# B&R Automation Studio project HealthCareDemo (part 4)

#### Types.typ
```iecst
TYPE
	Vis6D_typ : 	STRUCT
		Cmd : Vis6DCmd_typ;
		Par : Pars6D_typ;
		Status : Vis6DStatus_typ;
		TableData : VisTableData_typ;
		Limits : Vis6DLimits_typ;
	END_STRUCT;
	Vis6DCmd_typ : 	STRUCT
		ErrorReset : BOOL;
		Power : BOOL;
		AsmStop : BOOL;
		ShStop : BOOL;
		AsmHalt : BOOL;
		ShHalt : BOOL;
		AsmResume : BOOL;
		ShResume : BOOL;
		ShuttleID : UINT;
		RecoverShuttle : BOOL;
		MoveLinear : BOOL;
		MoveArc : BOOL;
		MoveShort : BOOL;
		MoveAsync : BOOL;
		Move6DOF : BOOL;
		AsmLevitation : BOOL;
		ShLevitation : BOOL;
		AsmBuffer : BOOL;
		ShBuffer : BOOL;
		Reboot : BOOL;
		ShRecover : BOOL;
	END_STRUCT;
	Vis6DStatus_typ : 	STRUCT
		AsmStatus : AsmStatus_typ;
		AllShuttlesFound : BOOL;
		StatusMessage : STRING[80];
		CurrentState : STRING[80];
		ErrorID : DINT;
		SelectedShuttleIDString : STRING[80];
		MovementActive : BOOL;
		ShuttleBuffer : VisShuttleBufferStatus_typ;
		ErrorText : STRING[80];
	END_STRUCT;
	VisShuttleBufferStatus_typ : 	STRUCT
		ShuttleID : UINT;
		State : STRING[80];
		NumberOfCommands : UINT;
	END_STRUCT;
	VisTableData_typ : 	STRUCT
		Async : VisAsyncTable_typ;
		ShuttleStatus : VisShuttleStatusTable_typ;
	END_STRUCT;
	VisAsyncTable_typ : 	STRUCT
		TargetXArray : ARRAY[0..rdiMAX_ASYNC_SHUTTLES_M1]OF REAL;
		TargetYArray : ARRAY[0..rdiMAX_ASYNC_SHUTTLES_M1]OF REAL;
		ShuttleIDArray : ARRAY[0..rdiMAX_ASYNC_SHUTTLES_M1]OF UINT;
	END_STRUCT;
	VisShuttleStatusTable_typ : 	STRUCT
		ShuttleID : ARRAY[0..MAX_NUM_SHUTTLES_M1]OF UINT;
		ShuttleIDString : ARRAY[0..MAX_NUM_SHUTTLES_M1]OF STRING[80];
		ShuttleStateText : ARRAY[0..MAX_NUM_SHUTTLES_M1]OF STRING[80];
		X : ARRAY[0..MAX_NUM_SHUTTLES_M1]OF REAL;
		Y : ARRAY[0..MAX_NUM_SHUTTLES_M1]OF REAL;
		Z : ARRAY[0..MAX_NUM_SHUTTLES_M1]OF REAL;
		Rx : ARRAY[0..MAX_NUM_SHUTTLES_M1]OF REAL;
		Ry : ARRAY[0..MAX_NUM_SHUTTLES_M1]OF REAL;
		Rz : ARRAY[0..MAX_NUM_SHUTTLES_M1]OF REAL;
	END_STRUCT;
END_TYPE

(*Insert your comment here.*)

TYPE
	Vis6DRealMinMax_typ : 	STRUCT
		Min : REAL;
		Max : REAL;
	END_STRUCT;
	Vis6DLimits_typ : 	STRUCT
		Linear : Vis6DLimitsLinear_typ;
		Arc : Vis6DLimitsArc_typ;
		Short : Vis6DLimitsShort_typ;
		SixDOF : Vis6DLimits6DOF_typ;
		Async : Vis6DLimitsAsync_typ;
	END_STRUCT;
	Vis6DLimitsLinear_typ : 	STRUCT
		X : Vis6DRealMinMax_typ;
		Y : Vis6DRealMinMax_typ;
		Velocity : Vis6DRealMinMax_typ;
		EndVelocity : Vis6DRealMinMax_typ;
		Acceleration : Vis6DRealMinMax_typ;
	END_STRUCT;
	Vis6DLimitsArc_typ : 	STRUCT
		AngleX : Vis6DRealMinMax_typ;
		AngleY : Vis6DRealMinMax_typ;
		Angle : Vis6DRealMinMax_typ;
		RadiusX : Vis6DRealMinMax_typ;
		RadiusY : Vis6DRealMinMax_typ;
		Radius : Vis6DRealMinMax_typ;
		Velocity : Vis6DRealMinMax_typ;
		EndVelocity : Vis6DRealMinMax_typ;
		Acceleration : Vis6DRealMinMax_typ;
	END_STRUCT;
	Vis6DLimitsShort_typ : 	STRUCT
		CenterX : Vis6DRealMinMax_typ;
		CenterY : Vis6DRealMinMax_typ;
		Z : Vis6DRealMinMax_typ;
		Rx : Vis6DRealMinMax_typ;
		Ry : Vis6DRealMinMax_typ;
		Rz : Vis6DRealMinMax_typ;
		VelZ : Vis6DRealMinMax_typ;
		VelRx : Vis6DRealMinMax_typ;
		VelRy : Vis6DRealMinMax_typ;
		VelRz : Vis6DRealMinMax_typ;
	END_STRUCT;
	Vis6DLimits6DOF_typ : 	STRUCT
		X : Vis6DRealMinMax_typ;
		Y : Vis6DRealMinMax_typ;
		Velocity : Vis6DRealMinMax_typ;
		Acceleration : Vis6DRealMinMax_typ;
		Z : Vis6DRealMinMax_typ;
		Rx : Vis6DRealMinMax_typ;
		Ry : Vis6DRealMinMax_typ;
		Rz : Vis6DRealMinMax_typ;
		VelZ : Vis6DRealMinMax_typ;
		VelRx : Vis6DRealMinMax_typ;
		VelRy : Vis6DRealMinMax_typ;
		VelRz : Vis6DRealMinMax_typ;
	END_STRUCT;
	Vis6DLimitsAsync_typ : 	STRUCT
		Velocity : Vis6DRealMinMax_typ;
		Acceleration : Vis6DRealMinMax_typ;
		X : Vis6DRealMinMax_typ;
		Y : Vis6DRealMinMax_typ;
	END_STRUCT;
END_TYPE
```

#### Variables.var
```iecst
VAR
	i : UINT;
	Core : rdi6DCore;
	Pars : Pars6D_typ;
	Vis : Vis6D_typ := (Limits:=(Linear:=(X:=(Min:=0.0,Max:=0.42),Y:=(Min:=0.0,Max:=0.18),Velocity:=(Min:=0.0,Max:=1.0),EndVelocity:=(Min:=0.0,Max:=1.0),Acceleration:=(Min:=0.0,Max:=10.0)),Arc:=(AngleX:=(Min:=0.0,Max:=0.42),AngleY:=(Min:=0.0,Max:=0.18),Angle:=(Min:=0.0,Max:=6.28319),RadiusX:=(Min:=0.0,Max:=0.42),RadiusY:=(Min:=0.0,Max:=0.18),Radius:=(Min:=0.0,Max:=0.1),Velocity:=(Min:=0.0,Max:=1.0),EndVelocity:=(Min:=0.0,Max:=1.0),Acceleration:=(Min:=0.0,Max:=10.0)),Short:=(CenterX:=(Min:=0.0,Max:=0.42),CenterY:=(Min:=0.0,Max:=0.18),Z:=(Min:=0.0,Max:=0.003),Rx:=(Min:=0.0,Max:=0.0872665),Ry:=(Min:=0.0,Max:=0.0872665),Rz:=(Min:=0.0,Max:=0.226893),VelZ:=(Min:=0.0,Max:=0.15),VelRx:=(Min:=0.0,Max:=0.1),VelRy:=(Min:=0.0,Max:=0.1),VelRz:=(Min:=0.0,Max:=0.3)),SixDOF:=(X:=(Min:=0.0,Max:=0.42),Y:=(Min:=0.0,Max:=0.18),Velocity:=(Min:=0.0,Max:=1.0),Acceleration:=(Min:=0.0,Max:=10.0),Z:=(Min:=0.0,Max:=0.003),Rx:=(Min:=0.0,Max:=0.0872665),Ry:=(Min:=0.0,Max:=0.0872665),Rz:=(Min:=0.0,Max:=0.226893),VelZ:=(Min:=0.0,Max:=0.15),VelRx:=(Min:=0.0,Max:=0.1),VelRy:=(Min:=0.0,Max:=0.1),VelRz:=(Min:=0.0,Max:=0.3)),Async:=(Velocity:=(Min:=0.0,Max:=1.0),Acceleration:=(Min:=0.0,Max:=10.0),X:=(Min:=0.0,Max:=0.42),Y:=(Min:=0.0,Max:=0.18))));
	TestStart : BOOL;
	ShState : McAcp6DShStateEnum;
	ShStatusTexts : ARRAY[0..15] OF STRING[80] := ['UNDETECTED','DISCOVERING','LANDED','IDLING','DISABLED','MOTION','WAIT','STOPPING','OBSTACLE','HOLD','STOPPED',3(''),'ERROR','RESERVED'];
	ShBufferStateTexts : ARRAY[0..1] OF STRING[80] := ['OPEN','BLOCKED'];
	StringPlacehold : STRING[80];
END_VAR
```

#### Main.st
```iecst
PROGRAM _INIT
	Core.Parameters := ADR(Pars);
	Core.AsmRef := ADR(g6dAssembly);
	Core.Enable := TRUE;
	ShState;
	TestStart := TRUE;

	Vis.Cmd.ShuttleID := 1;
	//

	Vis.Par.Linear.Position.X := 0.12;		// m
	Vis.Par.Linear.Position.Y := 0.12;		// m
	Vis.Par.Linear.Velocity := 1.0;			// m/s
	Vis.Par.Linear.EndVelocity := 0.0;		// m/s
	Vis.Par.Linear.Acceleration := 10.0;	// m/s^2

	Vis.Par.Arc.Radius.Position.X := 0.12;	// m
	Vis.Par.Arc.Radius.Position.Y := 0.12; // m
	Vis.Par.Arc.Radius.Radius := 0.0;		// m
	Vis.Par.Arc.Angular.Center.X := 0.12;	// m
	Vis.Par.Arc.Angular.Center.Y := 0.12;	// m
	Vis.Par.Arc.Angular.Angle := 0.0;		// rad
	Vis.Par.Arc.Velocity := 1.0;			// m/s
	Vis.Par.Arc.EndVelocity := 0.0;			// m/s
	Vis.Par.Arc.Acceleration := 10.0;		// m/s^2

	Vis.Par.ShortAxis.Rotation.Center.X := 0.18;	// m
	Vis.Par.ShortAxis.Rotation.Center.Y := 0.18;	// m
	Vis.Par.ShortAxis.Position.Z := 0.001;			// m
	Vis.Par.ShortAxis.Velocity.Z := 0.002;			// m/s
	Vis.Par.ShortAxis.Velocity.Rx := 0.0873;		// rad/s
	Vis.Par.ShortAxis.Velocity.Ry := 0.0873;		// rad/s
	Vis.Par.ShortAxis.Velocity.Rz := 0.0873;		// rad/s

	Vis.Par.SixDOF.InPlane.Position.X := 0.12;		// m
	Vis.Par.SixDOF.InPlane.Position.Y := 0.12;		// m
	Vis.Par.SixDOF.ShortAxis.Position.Z := 0.001;	// m
	Vis.Par.SixDOF.InPlane.Velocity := 1.0;			// m/s
	Vis.Par.SixDOF.InPlane.Acceleration := 10.0;	// m/s^2
	Vis.Par.SixDOF.ShortAxis.Velocity.Z := 0.002;	// m/s
	Vis.Par.SixDOF.ShortAxis.Velocity.Rx := 0.0873;	// rad/s
	Vis.Par.SixDOF.ShortAxis.Velocity.Ry := 0.0873;	// rad/s
	Vis.Par.SixDOF.ShortAxis.Velocity.Rz := 0.0873;	// rad/s

	Vis.Par.Async.Velocity := 0.5;		// m/s
	Vis.Par.Async.Acceleration := 5.0;	// m/s^2

END_PROGRAM

PROGRAM _CYCLIC
	(* Insert code here *)
	gFB;

	IF TestStart THEN
		Vis.Cmd.ShuttleID := STRING_TO_UINT(Vis.Status.SelectedShuttleIDString);

		Core.Power := Vis.Cmd.Power;
		Core.ShuttleID := Vis.Cmd.ShuttleID;
		Core.ErrorReset := Vis.Cmd.ErrorReset;

		Core.MoveLinear := Vis.Cmd.MoveLinear;
		Core.MoveArc := Vis.Cmd.MoveArc;
		Core.MoveShort := Vis.Cmd.MoveShort;
		Core.Move6DOF := Vis.Cmd.Move6DOF;
		Core.MoveAsync := Vis.Cmd.MoveAsync;

		Core.AsmStop := Vis.Cmd.AsmStop;
		Core.AsmHalt := Vis.Cmd.AsmHalt;
		Core.AsmResume := Vis.Cmd.AsmResume;

		Core.ShStop := Vis.Cmd.ShStop;
		Core.ShHalt := Vis.Cmd.ShHalt;
		Core.ShResume := Vis.Cmd.ShResume;

		Core.AsmLevitation := Vis.Cmd.AsmLevitation;
		Core.ShLevitation := Vis.Cmd.ShLevitation;
		Core.AsmBuffer := Vis.Cmd.AsmBuffer;
		Core.ShBuffer := Vis.Cmd.ShBuffer;

		Core.Reboot := Vis.Cmd.Reboot;
		Core.ShRecover := Vis.Cmd.ShRecover;

		FOR i := 0 TO rdiMAX_ASYNC_SHUTTLES_M1 DO
			Vis.Par.Async.ShuttleTable[i].ShuttleID := Vis.TableData.Async.ShuttleIDArray[i];
			Vis.Par.Async.ShuttleTable[i].X := Vis.TableData.Async.TargetXArray[i];
			Vis.Par.Async.ShuttleTable[i].Y := Vis.TableData.Async.TargetYArray[i];
		END_FOR

		FOR i := 0 TO MAX_NUM_SHUTTLES_M1 DO
			Vis.TableData.ShuttleStatus.ShuttleID[i] := Core.ShuttleArray[i].ShuttleID;

			Vis.TableData.ShuttleStatus.ShuttleIDString[i] := '{"value":"';
			StringPlacehold := UINT_TO_STRING(Core.ShuttleArray[i].ShuttleID);
			Vis.TableData.ShuttleStatus.ShuttleIDString[i] := CONCAT(Vis.TableData.ShuttleStatus.ShuttleIDString[i], StringPlacehold);
			Vis.TableData.ShuttleStatus.ShuttleIDString[i] := CONCAT(Vis.TableData.ShuttleStatus.ShuttleIDString[i], '","text":"');
			StringPlacehold := UINT_TO_STRING(Core.ShuttleArray[i].ShuttleID);
			Vis.TableData.ShuttleStatus.ShuttleIDString[i] := CONCAT(Vis.TableData.ShuttleStatus.ShuttleIDString[i], StringPlacehold);
			Vis.TableData.ShuttleStatus.ShuttleIDString[i] := CONCAT(Vis.TableData.ShuttleStatus.ShuttleIDString[i], '"}');

			Vis.TableData.ShuttleStatus.ShuttleStateText[i] := ShStatusTexts[Core.ShuttleArray[i].State];

			Vis.TableData.ShuttleStatus.X[i] := Core.ShuttleArray[i].Position.X;
			Vis.TableData.ShuttleStatus.Y[i] := Core.ShuttleArray[i].Position.Y;
			Vis.TableData.ShuttleStatus.Z[i] := Core.ShuttleArray[i].Position.Z;
			Vis.TableData.ShuttleStatus.Rx[i] := Core.ShuttleArray[i].Position.Rx;
			Vis.TableData.ShuttleStatus.Ry[i] := Core.ShuttleArray[i].Position.Ry;
			Vis.TableData.ShuttleStatus.Rz[i] := Core.ShuttleArray[i].Position.Rz;

		END_FOR

		brsmemcpy(ADR(Pars), ADR(Vis.Par), SIZEOF(Pars6D_typ));

		(* Copy Statuses *)
		brsmemcpy(ADR(Vis.Status.AsmStatus), ADR(Core.AsmStatus), SIZEOF(AsmStatus_typ));
		brsmemcpy(ADR(Vis.Status.StatusMessage), ADR(Core.StatusMessage), SIZEOF(Vis.Status.StatusMessage));
		brsmemcpy(ADR(Vis.Status.CurrentState), ADR(Core.CurrentState), SIZEOF(Vis.Status.CurrentState));

		Vis.Status.AllShuttlesFound := Core.AllShuttlesFound;
		Vis.Status.MovementActive := Core.MovementActive;
		Vis.Status.ErrorID := Core.ErrorID;

		Vis.Status.ShuttleBuffer.ShuttleID := Core.ShuttleBufferInfo.ShuttleID;
		Vis.Status.ShuttleBuffer.NumberOfCommands := Core.ShuttleBufferInfo.NumberOfCommands;
		Vis.Status.ShuttleBuffer.State := ShBufferStateTexts[Core.ShuttleBufferInfo.State];

		IF Core.Error THEN
			IF Core.ErrorID = -1065799680 THEN
				Vis.Status.ErrorText := 'Wrong shuttle state';
			ELSIF Core.ErrorID = -1065801966 THEN
				Vis.Status.ErrorText := 'The ACOPOS6D object is invalid';
			ELSE
				Vis.Status.ErrorText := 'Lookup ErrorID in the Help';
			END_IF
		ELSE
			Vis.Status.ErrorText := '';
		END_IF

	END_IF

	Core();

END_PROGRAM

PROGRAM _EXIT
	(* Insert code here *)

END_PROGRAM
```

### Program Logical/Source/Core/Main (IEC)

#### Types.typ
```iecst
TYPE
	MainSystemStatesEnum :
		(
		MAIN_OFF,
		MAIN_INIT,
		MAIN_RECOVERING,
		MAIN_READY,
		MAIN_STARTUP,
		MAIN_RUN_DEMO,
		MAIN_STOPPING,
		MAIN_ERROR,
		MAIN_RESET
		);
END_TYPE
```

#### Variables.var
```iecst
VAR
	state : MainSystemStatesEnum;
	errorState : MainSystemStatesEnum;
END_VAR
```

#### Cyclic.st
```iecst
PROGRAM _CYCLIC
	CASE state OF
		// ***************************** Getting Shuttles State
		MAIN_OFF:

			IF gSystemIf.Cmd.Power THEN
				gAcp6DIf.Cmd.Power := TRUE;

				state := MAIN_INIT;
			END_IF

		// ***************************** Initalization/Startup State
		MAIN_INIT:
			IF gAcp6DIf.Sts.Error THEN
				errorState := state;
				state := MAIN_ERROR;
			ELSIF gAcp6DIf.Sts.AssemblyReady THEN
				IF gStationsIf.Sts.RoutingInitalized THEN
					gStationsIf.Cmd.Enable := TRUE;

					IF gStationsIf.Sts.IncubatorActive THEN
						gStationsIf.Cmd.Recover := TRUE;
						state := MAIN_RECOVERING;
					END_IF
				END_IF
			END_IF
		// ***************************** Recovering State
		MAIN_RECOVERING:
			IF NOT gStationsIf.Cmd.Recover AND gStationsIf.Sts.PipetteActive[0] AND
				gStationsIf.Sts.PipetteActive[1] THEN

				//gSystemIf.Cmd.Run := TRUE;
				state := MAIN_READY;
			END_IF
		// ***************************** Ready State
		MAIN_READY:
			IF gSystemIf.Cmd.Run THEN
				gStationsIf.Cmd.Run := TRUE;

				state := MAIN_STARTUP;
			END_IF
		MAIN_STARTUP:
		//Startup, Send 1 shuttle to Analyzer, send 1 shuttle to Incubator

	END_CASE;

END_PROGRAM
```

#### Init.st
```iecst
PROGRAM _INIT
	gSysRecipe.DefaultVel := 0.5;
	gSysRecipe.DefaultAccel := 5;
	gSysRecipe.DefaultWaitTime := 1000;

	gStationsIf.Par.Incubator.Waypoint := WP_1;
END_PROGRAM
```

### Program Logical/Source/Core/Acp6DCtrl (IEC)

#### Types.typ
```iecst
TYPE
	Acp6DFbsTyp : 	STRUCT
		PowerOnFb : MC_BR_AsmPowerOn_Acp6D;
		PowerOfFb : MC_BR_AsmPowerOff_Acp6D;
		AsmGetShuttleFb : MC_BR_AsmGetShuttle_Acp6D;
		MoveAsyncFb : MC_BR_MoveInPlaneAsync_Acp6D;
		AsmStatusFb : MC_BR_AsmReadStatus_Acp6D;
		AsmInfoFb : MC_BR_AsmGetInfo_Acp6D;
	END_STRUCT;
	Acp6DStateEnum :
		(
		ACP6D_IDLE,
		ACP6D_POWER_ON,
		ACP6D_GET_SHUTTLE,
		ACP6D_NEXT_SHUTTLE,
		ACP6D_MOVE_STARTUP,
		ACP6D_OPERATIONAL,
		ACP6D_POWER_OFF,
		ACP6D_ERROR,
		ACP6D_RESET
		);
END_TYPE
```

#### Variables.var
```iecst
VAR
	state : Acp6DStateEnum;
	fbs : Acp6DFbsTyp;
	errorState : Acp6DStateEnum;
	i : UINT;
	testFb : MC_BR_MoveInPlaneAsync_Acp6D;
END_VAR
```

#### Cyclic.st
```iecst
PROGRAM _CYCLIC
	gAcp6DIf.Sts.AssemblyInfo := fbs.AsmInfoFb.AssemblyInfo;
	gAcp6DIf.Sts.AssemblyDisabled := fbs.AsmStatusFb.AssemblyDisabled;
	gAcp6DIf.Sts.AssemblyReady := fbs.AsmStatusFb.AssemblyReady;
	gAcp6DIf.Sts.AssemblyHoming := fbs.AsmStatusFb.AssemblyHoming;
	gAcp6DIf.Sts.AssemblyStopping := fbs.AsmStatusFb.AssemblyStopping;
	gAcp6DIf.Sts.AssemblyStartup:= fbs.AsmStatusFb.AssemblyStartUp;
	gAcp6DIf.Sts.AssemblyErrorStop := fbs.AsmStatusFb.AssemblyErrorStop;
	fbs.AsmStatusFb.Assembly := ADR(gAcp6DIf.Par.Asm);
	fbs.AsmStatusFb.Enable := TRUE;

	fbs.AsmInfoFb.Assembly := ADR(gAcp6DIf.Par.Asm);
	fbs.AsmInfoFb.Execute := TRUE AND NOT gAcp6DIf.Cmd.ResetInfo;

	CASE state OF
		// ***************************** Idle State
		ACP6D_IDLE:
			IF gAcp6DIf.Sts.AssemblyReady THEN
				fbs.PowerOfFb.Assembly := ADR(gAcp6DIf.Par.Asm);
				fbs.PowerOfFb.Execute := TRUE;

				state := ACP6D_POWER_OFF;
			ELSIF gAcp6DIf.Cmd.Power AND gAcp6DIf.Sts.AssemblyDisabled THEN
				fbs.PowerOnFb.Assembly := ADR(gAcp6DIf.Par.Asm);
				fbs.PowerOnFb.Execute := TRUE;

				state := ACP6D_POWER_ON;
			END_IF

		// ***************************** Power On State
		ACP6D_POWER_ON:
			IF fbs.PowerOnFb.Error THEN
				gAcp6DIf.Sts.Error := TRUE;
				errorState := state;

				state := ACP6D_ERROR;
			ELSIF fbs.PowerOnFb.Done THEN
				fbs.PowerOnFb.Execute := FALSE;

				fbs.AsmGetShuttleFb.Assembly := ADR(gAcp6DIf.Par.Asm);
				fbs.AsmGetShuttleFb.Enable := TRUE;

				//Reset all the info in the interfaces

				brsmemset(ADR(gShIfs),0,NUM_SHUTTLES * SIZEOF(gShIfs[0]));

				state := ACP6D_GET_SHUTTLE;
			END_IF

		// ***************************** Getting Shuttles State
		ACP6D_GET_SHUTTLE:
			IF fbs.AsmGetShuttleFb.Error THEN
				gAcp6DIf.Sts.Error := TRUE;
				errorState := state;

				state := ACP6D_ERROR;
			ELSIF fbs.AsmGetShuttleFb.Valid THEN
				gShIfs[fbs.AsmGetShuttleFb.TotalCount - (fbs.AsmGetShuttleFb.RemainingCount + 1)].Cfg.Shuttle := fbs.AsmGetShuttleFb.Shuttle;
				gShIfs[fbs.AsmGetShuttleFb.TotalCount - (fbs.AsmGetShuttleFb.RemainingCount + 1)].Cfg.ID := fbs.AsmGetShuttleFb.AdditionalInfo.ShuttleID;
				gShIfs[fbs.AsmGetShuttleFb.TotalCount - (fbs.AsmGetShuttleFb.RemainingCount + 1)].Sts.Available := TRUE;
				IF fbs.AsmGetShuttleFb.RemainingCount > 0 THEN
					fbs.AsmGetShuttleFb.Next := TRUE;
					state := ACP6D_NEXT_SHUTTLE;
				ELSE
					fbs.AsmGetShuttleFb.Enable := FALSE;

					fbs.MoveAsyncFb.Assembly := ADR(gAcp6DIf.Par.Asm);
					FOR i := 0 TO gAcp6DIf.Sts.AssemblyInfo.NumberOfShuttles - 1 DO
	  					gSysRecipe.StartupPars.MoveAsyncPars.AsyncPar[i].Shuttle := ADR(gShIfs[i].Cfg.Shuttle);
					END_FOR;
					fbs.MoveAsyncFb.Parameters := gSysRecipe.StartupPars.MoveAsyncPars;

					//fbs.MoveAsyncFb.Execute := TRUE;
					state := ACP6D_OPERATIONAL; //No longer need this when using Routing Library
				END_IF
			END_IF

		// ***************************** Find Next Shuttle State
		ACP6D_NEXT_SHUTTLE:
			IF fbs.AsmGetShuttleFb.Error THEN
				gAcp6DIf.Sts.Error := TRUE;
				errorState := state;

				state := ACP6D_ERROR;
			ELSIF fbs.AsmGetShuttleFb.Valid THEN
				fbs.AsmGetShuttleFb.Next := FALSE;

				state := ACP6D_GET_SHUTTLE;
			END_IF
		// ***************************** Move to Startup Positions State
		ACP6D_MOVE_STARTUP:
			IF fbs.MoveAsyncFb.Error THEN
				gAcp6DIf.Sts.Error := TRUE;
				errorState := state;

				state := ACP6D_ERROR;
			ELSIF fbs.MoveAsyncFb.Done THEN
				fbs.MoveAsyncFb.Execute := FALSE;

				state := ACP6D_OPERATIONAL;
			END_IF
		// ***************************** Operational State
		ACP6D_OPERATIONAL:
			IF NOT gAcp6DIf.Cmd.Power THEN
				fbs.PowerOfFb.Assembly := ADR(gAcp6DIf.Par.Asm);
				fbs.PowerOfFb.Execute := TRUE;

				state := ACP6D_POWER_OFF;
			END_IF

		// ***************************** Powering Off State
		ACP6D_POWER_OFF:
			IF fbs.PowerOfFb.Error THEN
				gAcp6DIf.Sts.Error := TRUE;
				errorState := state;

				state := ACP6D_ERROR;
			ELSIF fbs.PowerOfFb.Done THEN
				fbs.PowerOfFb.Execute := FALSE;
				brsmemset(ADR(gShIfs),0,NUM_SHUTTLES * SIZEOF(gShIfs[0]));

				state := ACP6D_IDLE;
			END_IF

		// ***************************** Error State
		ACP6D_ERROR:
			IF gAcp6DIf.Cmd.Reset THEN
				state := ACP6D_RESET;
			END_IF

		// ***************************** Restting State
		ACP6D_RESET:
			fbs.AsmGetShuttleFb.Enable := FALSE;
			fbs.AsmGetShuttleFb.Next := FALSE;
			fbs.MoveAsyncFb.Execute := FALSE;
			fbs.MoveAsyncFb.Execute := FALSE;
			fbs.PowerOnFb.Execute := FALSE;
			fbs.PowerOfFb.Execute := FALSE;

			gAcp6DIf.Sts.Error := FALSE;

			state := ACP6D_IDLE;
	END_CASE;

	fbs.AsmInfoFb();
	fbs.PowerOnFb();
	fbs.PowerOfFb();
	fbs.AsmGetShuttleFb();
	fbs.MoveAsyncFb();
	fbs.AsmStatusFb();

END_PROGRAM
```

#### Init.st
```iecst
PROGRAM _INIT
	gFB;
	gAcp6DIf.Par.Asm := g6dAssembly;

	gSysRecipe.StartupPars.MoveAsyncPars.Velocity := 1.0;
	gSysRecipe.StartupPars.MoveAsyncPars.Acceleration := 10.0;
	gSysRecipe.StartupPars.MoveAsyncPars.AsyncPar[0].X := 0.060;
	gSysRecipe.StartupPars.MoveAsyncPars.AsyncPar[0].Y := 0.060;
	gSysRecipe.StartupPars.MoveAsyncPars.AsyncPar[1].X := 0.060;
	gSysRecipe.StartupPars.MoveAsyncPars.AsyncPar[1].Y := 0.060;
	gSysRecipe.StartupPars.MoveAsyncPars.AsyncPar[2].X := 0.360;
	gSysRecipe.StartupPars.MoveAsyncPars.AsyncPar[2].Y := 0.120;
END_PROGRAM
```

### Program Logical/Source/Core/Program (IEC)

#### Types.typ
```iecst
TYPE
	FbsTyp : 	STRUCT
		MoveAsyncFb : MC_BR_MoveInPlaneAsync_Acp6D;
		HelpMoveFb : Acp6DMoveBlockFb;
	END_STRUCT;
END_TYPE
```

#### Variables.var
```iecst
VAR
	state : INT;
	test : BOOL;
	fbs : FbsTyp;
	pars : ARRAY[0..9] OF Acp6DMoveListTyp;
END_VAR
```

#### Cyclic.st
```iecst
PROGRAM _CYCLIC
	//Move all shuttles to some start location
	//Leave one shuttle to just run through a handful of movements repeatedly
	//Route all the other shuttles to mix up their locations

	gSystemIf;
	CASE state OF
		0:
			IF test THEN
				fbs.MoveAsyncFb.Assembly := ADR(g6dAssembly);
				fbs.MoveAsyncFb.Parameters.AsyncPar[0].Shuttle := ADR(gShIfs[0].Cfg.Shuttle);
				fbs.MoveAsyncFb.Parameters.AsyncPar[0].X := 0.060;
				fbs.MoveAsyncFb.Parameters.AsyncPar[0].Y := 0.180;
				fbs.MoveAsyncFb.Parameters.AsyncPar[1].Shuttle := ADR(gShIfs[1].Cfg.Shuttle);
				fbs.MoveAsyncFb.Parameters.AsyncPar[1].X := 0.06;
				fbs.MoveAsyncFb.Parameters.AsyncPar[1].Y := 0.06;
				fbs.MoveAsyncFb.Parameters.AsyncPar[2].Shuttle := ADR(gShIfs[2].Cfg.Shuttle);
				fbs.MoveAsyncFb.Parameters.AsyncPar[2].X := 0.36;
				fbs.MoveAsyncFb.Parameters.AsyncPar[2].Y := 0.12;
				fbs.MoveAsyncFb.Parameters.Velocity := 0.25;
				fbs.MoveAsyncFb.Parameters.MoveOnlySelectedShuttles := FALSE;
				fbs.MoveAsyncFb.Parameters.Acceleration := 1.0;
				fbs.MoveAsyncFb.Execute := TRUE;

				state := 10;
			END_IF
		10:
			IF fbs.MoveAsyncFb.Done THEN
				fbs.MoveAsyncFb.Execute := FALSE;

				state := 11;
			END_IF
		11:
			pars[0].MoveType := acp6d_MOVE_ARC;
			pars[0].Arc.Velocity := 0.05;
			pars[0].Arc.Acceleration := 1;
			pars[0].Arc.EndVelocity := 0;
			pars[0].Arc.Mode := mcACP6D_MOVE_RELATIVE;
			pars[0].Arc.Option := mcACP6D_ARC_ANGULAR;
			pars[0].Arc.Angular.Center.X := 0.005;
			pars[0].Arc.Angular.Center.Y := 0.0000;
			pars[0].Arc.Direction := mcACP6D_ARC_CLOCKWISE;
			pars[0].Arc.Angular.Angle := 3.1415 * 2 * 40;

			fbs.HelpMoveFb.Shuttle := gShIfs[2].Cfg.Shuttle;
			fbs.HelpMoveFb.Pars.NumMoves := 1;
			fbs.HelpMoveFb.Pars.MoveList := ADR(pars);
			fbs.HelpMoveFb.Execute := TRUE;

			state := 20;
		20:
			fbs.MoveAsyncFb.Assembly := ADR(g6dAssembly);
			fbs.MoveAsyncFb.Parameters.AsyncPar[0].Shuttle := ADR(gShIfs[0].Cfg.Shuttle);
			fbs.MoveAsyncFb.Parameters.AsyncPar[0].X := 0.180;
			fbs.MoveAsyncFb.Parameters.AsyncPar[0].Y := 0.42;
			fbs.MoveAsyncFb.Parameters.AsyncPar[1].Shuttle := ADR(gShIfs[1].Cfg.Shuttle);
			fbs.MoveAsyncFb.Parameters.AsyncPar[1].X := 0.06;
			fbs.MoveAsyncFb.Parameters.AsyncPar[1].Y := 0.42;
			fbs.MoveAsyncFb.Parameters.AsyncPar[2].Shuttle := 0;
			fbs.MoveAsyncFb.Parameters.AsyncPar[2].X := 0;
			fbs.MoveAsyncFb.Parameters.AsyncPar[2].Y := 0;
			fbs.MoveAsyncFb.Parameters.Acceleration := 1.0;
			fbs.MoveAsyncFb.Parameters.Velocity := 0.25;
			fbs.MoveAsyncFb.Parameters.MoveOnlySelectedShuttles := TRUE;
			fbs.MoveAsyncFb.Execute := TRUE;
			state := 21;
		21:
			IF fbs.MoveAsyncFb.Done THEN
				fbs.MoveAsyncFb.Execute := FALSE;

				state := 22;
			END_IF
		22:
			fbs.MoveAsyncFb.Parameters.AsyncPar[0].Shuttle := ADR(gShIfs[0].Cfg.Shuttle);
			fbs.MoveAsyncFb.Parameters.AsyncPar[0].X := 0.060;
			fbs.MoveAsyncFb.Parameters.AsyncPar[0].Y := 0.06;
			fbs.MoveAsyncFb.Parameters.AsyncPar[1].Shuttle := ADR(gShIfs[1].Cfg.Shuttle);
			fbs.MoveAsyncFb.Parameters.AsyncPar[1].X := 0.36;
			fbs.MoveAsyncFb.Parameters.AsyncPar[1].Y := 0.36;
			fbs.MoveAsyncFb.Parameters.Acceleration := 1.0;
			fbs.MoveAsyncFb.Parameters.Velocity := 0.25;
			fbs.MoveAsyncFb.Parameters.MoveOnlySelectedShuttles := TRUE;
			fbs.MoveAsyncFb.Execute := TRUE;
			state := 30;

	END_CASE;

	fbs.HelpMoveFb();
	fbs.MoveAsyncFb();

END_PROGRAM
```

### Program Logical/Source/Core/RoutingDefinitions (ANSIC)

#### Types.typ
```iecst
TYPE
	RoutingDefineEnum :
		(
		DEF_IDLE,
		DEF_INIT_ROUTER,
		DEF_INIT_ENTRY_PATHS,
		DEF_INIT_EXIT_PATHS,
		DEF_INIT_DESTINATIONS,
		DEF_INIT_RECOVERY_POINTS,
		DEF_INIT_WAYPOINTS,
		DEF_CHECK_WAYPOINT_DESTS,
		DEF_LINK_WAYPOINTS_TO_DESTS,
		DEF_LINK_WAYPOINTS_TO_WAYPOINTS,
		DEF_DONE,
		DEF_ADD_SHUTTLES,
		DEF_READY,
		DEF_RECOVERY,
		DEF_SEND_TO_START,
		DEF_RUNNING,
		DEF_ERROR
		);
	InitFbsTyp : 	STRUCT
		routerFb : rl6dRouterMan;
		addPathFb : rl6dRouterAddPathFromData;
		addRecPointFb : rl6dDestAddRecoveryPosFromData;
		createDestFb : rl6dRouterAddDestination;
		createWaypointFb : rl6dRouterAddWaypoint;
		linkWaypointFb : rl6dWaypointSetNextWaypoint;
		linkWayPointDestFb : rl6dWaypointAddDestination;
		addShToRouter : rl6dRouterAddShFromAsm;
		recoverFb : rl6dRouterExecuteRecovery;
	END_STRUCT;
END_TYPE
```

#### Variables.var
```iecst
VAR CONSTANT
	numDestinations : USINT := 6;
	numWaypoints : USINT := 5;
END_VAR
VAR
	state : RoutingDefineEnum;
	fbs : InitFbsTyp;
	Init : BOOL;
	j : USINT;
	i : USINT;
END_VAR
```

#### Cyclic.c
```c
#include <bur/plctypes.h>

#ifdef _DEFAULT_INCLUDES
#include <AsDefault.h>
#endif
#define TRUE 1
#define FALSE 0

void _CYCLIC ProgramCyclic(void)
{
	//On Command: Initalize the configuration for the routing library
	switch (state)
	{
		case DEF_IDLE:
			if(Init || gAcp6DIf.Sts.AssemblyReady){
				fbs.routerFb.Assembly = &g6dAssembly;
				fbs.routerFb.UserDataSize = sizeof(UserDataType);
				fbs.routerFb.Enable = TRUE;

				//Starting from 1 because the 0 index is going to be the "emtpy or default" index for most items
				i = 1;

				state = DEF_INIT_ROUTER;
			}
			break;
		case DEF_INIT_ROUTER:
			if(fbs.routerFb.Error){

			}
			else if(fbs.routerFb.Active){
				fbs.addPathFb.Router = &fbs.routerFb.Router;
				fbs.addPathFb.DataAddress = &gDests[i].Entry.PathPoints;
				fbs.addPathFb.DataSize = sizeof(gDests[i].Entry.PathPoints[0]) * gDests[i].Entry.Length;
				brsstrcpy(&fbs.addPathFb.Name,&gDests[i].Entry.Name);
				fbs.addPathFb.Execute = TRUE;

				state = DEF_INIT_ENTRY_PATHS;
			}
			break;
		case DEF_INIT_ENTRY_PATHS:
			if(fbs.addPathFb.Error){
				state = DEF_ERROR;
			}
			else if(fbs.addPathFb.Done){
				gDests[i].Entry.Path = fbs.addPathFb.Path;
				fbs.addPathFb.Execute = FALSE;

				i++;
				if(i > numDestinations){
					i = 1;

					fbs.addPathFb.DataAddress = &gDests[i].Exit.PathPoints;
					fbs.addPathFb.DataSize = sizeof(gDests[i].Exit.PathPoints[0]) * gDests[i].Exit.Length;
					brsstrcpy(&fbs.addPathFb.Name,&gDests[i].Exit.Name);

					state = DEF_INIT_EXIT_PATHS;
				}
				else{
					fbs.addPathFb.DataAddress = &gDests[i].Entry.PathPoints;
					fbs.addPathFb.DataSize = sizeof(gDests[i].Entry.PathPoints[0]) * gDests[i].Entry.Length;
					brsstrcpy(&fbs.addPathFb.Name,&gDests[i].Entry.Name);
				}

			}
			else{
				fbs.addPathFb.Execute = TRUE;
			}
			break;
		case DEF_INIT_EXIT_PATHS:
			if(fbs.addPathFb.Error){
				state = DEF_ERROR;
			}
			else if(fbs.addPathFb.Done){
				gDests[i].Exit.Path = fbs.addPathFb.Path;
				fbs.addPathFb.Execute = FALSE;

				i++;
				if(i > numDestinations){
					i = 0;

					fbs.createDestFb.Router = &fbs.routerFb.Router;
					if(gDests[i].Entry.Path.Ident != 0)
						fbs.createDestFb.EntryPath = &gDests[i].Entry.Path;
					if(gDests[i].Exit.Path.Ident != 0)
					fbs.createDestFb.ExitPath = &gDests[i].Exit.Path;
					fbs.createDestFb.Position = gDests[i].Position;
					brsstrcpy(&fbs.createDestFb.Name,&gDests[i].StationName);
					fbs.createDestFb.Execute = TRUE;

					state = DEF_INIT_DESTINATIONS;
				}
				else{
					fbs.addPathFb.DataAddress = &gDests[i].Exit.PathPoints;
					fbs.addPathFb.DataSize = sizeof(gDests[i].Exit.PathPoints[0]) * gDests[i].Exit.Length;
					brsstrcpy(&fbs.addPathFb.Name,&gDests[i].Exit.Name);
				}

			}
			else{
				fbs.addPathFb.Execute = TRUE;
			}
			break;
		case DEF_INIT_DESTINATIONS:
			if(fbs.createDestFb.Error){
				state = DEF_ERROR;
			}
			else if(fbs.createDestFb.Done){
				gDests[i].Destination = fbs.createDestFb.Destination;
				fbs.createDestFb.Execute = FALSE;

				i++;
				//Check to see if we've gone through all destinations
				if(i > numDestinations){
					i = 0;

					//Setup the recovery points
					fbs.addRecPointFb.Destination = &gDests[i].Destination;
					fbs.addRecPointFb.DataAddress = &gDests[i].RecoveryPts;
					fbs.addRecPointFb.DataSize = sizeof(gDests[i].RecoveryPts);
					fbs.addRecPointFb.Execute = TRUE;

					state = DEF_INIT_RECOVERY_POINTS;
				}
				else{
					//Haven't finished the destinations, so configure to complete the next destination
					fbs.createDestFb.Router = &fbs.routerFb.Router;
					fbs.createDestFb.EntryPath = &gDests[i].Entry.Path;
					fbs.createDestFb.ExitPath = &gDests[i].Exit.Path;
					fbs.createDestFb.Position = gDests[i].Position;
					brsstrcpy(&fbs.createDestFb.Name,&gDests[i].StationName);
				}

			}
			else{
				//Re-execute the block to handle the new parameter set
				fbs.createDestFb.Execute = TRUE;
			}
			break;
		case DEF_INIT_RECOVERY_POINTS:
			if(fbs.addRecPointFb.Error){
				state = DEF_ERROR;
			}
			else if(fbs.addRecPointFb.Done){
				fbs.addRecPointFb.Execute = FALSE;

				i++;
				//Check to see if we've gone through all destinations
				if(i > numDestinations){
					i = 1;

					//Setup the waypoints
					fbs.createWaypointFb.Router = &fbs.routerFb.Router;
					fbs.createWaypointFb.Position = gWps[i].Position;
					brsstrcpy(&fbs.createWaypointFb.Name,&gWps[i].Name);
					fbs.createWaypointFb.Execute = TRUE;

					state = DEF_INIT_WAYPOINTS;
				}
				else{
					//Haven't finished the recovery points, so configure to complete the next destination
					fbs.addRecPointFb.Destination = &gDests[i].Destination;
					fbs.addRecPointFb.DataAddress = &gDests[i].RecoveryPts;
					fbs.addRecPointFb.DataSize = sizeof(gDests[i].RecoveryPts);
				}

			}
			else{
				//Re-execute the block to handle the new parameter set
				fbs.addRecPointFb.Execute = TRUE;
			}
			break;
		case DEF_INIT_WAYPOINTS:
			if(fbs.createWaypointFb.Error){
				state = DEF_ERROR;
			}
			else if(fbs.createWaypointFb.Done){
				gWps[i].Waypoint = fbs.createWaypointFb.Waypoint;
				fbs.createWaypointFb.Execute = FALSE;

				i++;
				//Check to see if we've gone through all waypoints
				if(i > numWaypoints){
					i = 1;
					j = 0;

					if(gWps[i].Destinations[j] != DEST_DEFAULT){
						//We have, so now we need to add all destinations for each waypoint
						fbs.linkWayPointDestFb.Destination = &gDests[gWps[i].Destinations[j]].Destination;
						fbs.linkWayPointDestFb.Waypoint = &gWps[i].Waypoint;
						fbs.linkWayPointDestFb.Execute = TRUE;

						state = DEF_LINK_WAYPOINTS_TO_DESTS;
					}
					else{
						i++;
						state = DEF_LINK_WAYPOINTS_TO_DESTS;
					}
				}
				else{
					//Haven't finished the waypoints, so configure to complete the next waypoint
					fbs.createWaypointFb.Router = &fbs.routerFb.Router;
					fbs.createWaypointFb.Position = gWps[i].Position;
					brsstrcpy(&fbs.createWaypointFb.Name,gWps[i].Name);
				}

			}
			else{
				//Re-execute the block to handle the new parameter set
				fbs.createWaypointFb.Execute = TRUE;
			}
			break;
		case DEF_CHECK_WAYPOINT_DESTS:
			//Check to see if we've finished iterating through all waypoints
			if(i > numWaypoints){
				//We're done, move onto the next init state
				i = 1;
				j = 0;
				fbs.linkWaypointFb.Waypoint = &gWps[i].Waypoint;
				fbs.linkWaypointFb.NextWaypoint = &gWps[gWps[i].NextWaypoint].Waypoint;
				fbs.linkWaypointFb.Execute = TRUE;

				state = DEF_LINK_WAYPOINTS_TO_WAYPOINTS;
			}
			else{
				//Check to see if the next destination is defined
				if(gWps[i].Destinations[j] != DEST_DEFAULT && j < 6){ //Added 5 here as that's the current size (6) of the array. This is a temp fix
					//The destination has been defined let's add it now
					fbs.linkWayPointDestFb.Destination = &gDests[gWps[i].Destinations[j]].Destination;
					fbs.linkWayPointDestFb.Waypoint = &gWps[i].Waypoint;
					fbs.linkWayPointDestFb.Execute = TRUE;

					state = DEF_LINK_WAYPOINTS_TO_DESTS;
				}
				else{
					//The destination is not defined, we therefore are done with this waypoint
					i++;
					j = 0;
				}
			}
			break;
		case DEF_LINK_WAYPOINTS_TO_DESTS:
			if(fbs.linkWayPointDestFb.Error){
				state = DEF_ERROR;
			}
			else if(fbs.linkWayPointDestFb.Done){
				fbs.linkWayPointDestFb.Execute = FALSE;
				j++;
				state = DEF_CHECK_WAYPOINT_DESTS;
			}
			break;
		case DEF_LINK_WAYPOINTS_TO_WAYPOINTS:
			if(fbs.linkWaypointFb.Error){
				state = DEF_ERROR;
			}
			else if(fbs.linkWaypointFb.Done){
				fbs.linkWaypointFb.Execute = FALSE;

				i++;
				//Check to see if we've gone through all waypoints
				if(i > numWaypoints){
					i = 1;
					//We're all done!
					state = DEF_DONE;
				}
				else{
					//Haven't finished the waypoints, so configure to complete the next waypoint
					fbs.linkWaypointFb.Waypoint = &gWps[i].Waypoint;
					fbs.linkWaypointFb.NextWaypoint = &gWps[gWps[i].NextWaypoint].Waypoint;
				}

			}
			else{
				//Re-execute the block to handle the new parameter set
				fbs.linkWaypointFb.Execute = TRUE;
			}
			break;
		case DEF_DONE:
			gStationsIf.Sts.RoutingInitalized = TRUE;

			Init = FALSE;
			if(gAcp6DIf.Sts.AssemblyReady){

				fbs.addShToRouter.Router = &fbs.routerFb.Router;
				fbs.addShToRouter.Execute = TRUE;

				state = DEF_ADD_SHUTTLES;
			}
			break;
		case DEF_ADD_SHUTTLES:
			if(fbs.addShToRouter.Error){
			}
			else if(fbs.addShToRouter.Done){
				fbs.addShToRouter.Execute = FALSE;
				state = DEF_READY;
			}
			break;
		case DEF_READY:
			fbs.recoverFb.Velocity = 1.0;
			fbs.recoverFb.Acceleration = 10.0;
			fbs.recoverFb.Router = &fbs.routerFb.Router;
			if(gStationsIf.Cmd.Recover){
				fbs.recoverFb.Execute = TRUE;
				state = DEF_RECOVERY;
			}
			break;
		case DEF_RECOVERY:
			if(fbs.recoverFb.Done){
				fbs.recoverFb.Execute = FALSE;
				gStationsIf.Cmd.Recover = FALSE;

				state = DEF_RUNNING;
			}
			break;
		case DEF_RUNNING:
			break;
		case DEF_ERROR:
			break;
	}
	rl6dRouterMan(&fbs.routerFb);
	rl6dRouterAddPathFromData(&fbs.addPathFb);
	rl6dRouterAddDestination(&fbs.createDestFb);
	rl6dRouterAddWaypoint(&fbs.createWaypointFb);
	rl6dWaypointAddDestination(&fbs.linkWayPointDestFb);
	rl6dWaypointSetNextWaypoint(&fbs.linkWaypointFb);
	rl6dRouterAddShFromAsm(&fbs.addShToRouter);
	rl6dDestAddRecoveryPosFromData(&fbs.addRecPointFb);
	rl6dRouterExecuteRecovery(&fbs.recoverFb);
}
```

#### Init.c
```c
#include <bur/plctypes.h>

#ifdef _DEFAULT_INCLUDES
	#include <AsDefault.h>
#endif
#define TRUE 1
#define FALSE 0

void _INIT ProgramInit(void)
{
	//Define the destinations & their paths

	//*******Default Destination
	brsstrcpy(&gDests[DEST_DEFAULT].StationName,&"Default");
	gDests[DEST_DEFAULT].Position.X = 0.18;
	gDests[DEST_DEFAULT].Position.Y = 0.18;
	gDests[DEST_DEFAULT].RecoveryPts.X = 0.18;
	gDests[DEST_DEFAULT].RecoveryPts.Y = 0.18;

	//*******Incubator Destination
	brsstrcpy(&gDests[DEST_INCUBATOR].StationName,&"Incubator");
	gDests[DEST_INCUBATOR].Position.X = 0.06;
	gDests[DEST_INCUBATOR].Position.Y = 0.06;
	gDests[DEST_INCUBATOR].RecoveryPts.X = 0.06;
	gDests[DEST_INCUBATOR].RecoveryPts.Y = 0.06;

	brsstrcpy(&gDests[DEST_INCUBATOR].Entry.Name,&"Incubator Entry");
	gDests[DEST_INCUBATOR].Entry.PathPoints[0].X = 0.18;
	gDests[DEST_INCUBATOR].Entry.PathPoints[0].Y = 0.3;
	gDests[DEST_INCUBATOR].Entry.PathPoints[1].X = 0.18;
	gDests[DEST_INCUBATOR].Entry.PathPoints[1].Y = 0.06;
	gDests[DEST_INCUBATOR].Entry.Length = 2;

	brsstrcpy(&gDests[DEST_INCUBATOR].Exit.Name,&"Incubator Exit");
	gDests[DEST_INCUBATOR].Exit.PathPoints[0].X = 0.06;
	gDests[DEST_INCUBATOR].Exit.PathPoints[0].Y = 0.42;
	gDests[DEST_INCUBATOR].Exit.Length = 1;

	//******Analyzer Destination
	brsstrcpy(&gDests[DEST_ANALYZER].StationName,&"Analyzer");
	gDests[DEST_ANALYZER].Position.X = 0.06;
	gDests[DEST_ANALYZER].Position.Y = 0.66;
	gDests[DEST_ANALYZER].RecoveryPts.X = 0.06;
	gDests[DEST_ANALYZER].RecoveryPts.Y = 0.66;

	brsstrcpy(&gDests[DEST_ANALYZER].Entry.Name,&"Analyzer Entry");
	gDests[DEST_ANALYZER].Entry.PathPoints[0].X = 0.06;
	gDests[DEST_ANALYZER].Entry.PathPoints[0].Y = 0.30;
	gDests[DEST_ANALYZER].Entry.Length = 1;

	brsstrcpy(&gDests[DEST_ANALYZER].Exit.Name,&"Analyzer Exit");
	gDests[DEST_ANALYZER].Exit.PathPoints[0].X = 0.18;
	gDests[DEST_ANALYZER].Exit.PathPoints[0].Y = 0.66;
	gDests[DEST_ANALYZER].Exit.PathPoints[1].X = 0.18;
	gDests[DEST_ANALYZER].Exit.PathPoints[1].Y = 0.42;
	gDests[DEST_ANALYZER].Exit.Length = 2;

	//******Pipette 1 Destination
	brsstrcpy(&gDests[DEST_PIPETTE_1].StationName,&"Pipette 1");
	gDests[DEST_PIPETTE_1].Position.X = 0.36;
	gDests[DEST_PIPETTE_1].Position.Y = 0.60;
	gDests[DEST_PIPETTE_1].RecoveryPts.X = 0.36;
	gDests[DEST_PIPETTE_1].RecoveryPts.Y = 0.60;

	brsstrcpy(&gDests[DEST_PIPETTE_1].Entry.Name,&"Pipette 1 Entry");
	gDests[DEST_PIPETTE_1].Entry.PathPoints[0].X = 0.30;
	gDests[DEST_PIPETTE_1].Entry.PathPoints[0].Y = 0.60;
	gDests[DEST_PIPETTE_1].Entry.Length = 1;

	brsstrcpy(&gDests[DEST_PIPETTE_1].Exit.Name,&"Pipette 1 Exit");
	gDests[DEST_PIPETTE_1].Exit.PathPoints[0].X = 0.42;
	gDests[DEST_PIPETTE_1].Exit.PathPoints[0].Y = 0.60;
	gDests[DEST_PIPETTE_1].Exit.Length = 1;

	//******Pipette 2 Destination
	brsstrcpy(&gDests[DEST_PIPETTE_2].StationName,&"Pipette 2");
	gDests[DEST_PIPETTE_2].Position.X = 0.36;
	gDests[DEST_PIPETTE_2].Position.Y = 0.12;
	gDests[DEST_PIPETTE_2].RecoveryPts.X = 0.36;
	gDests[DEST_PIPETTE_2].RecoveryPts.Y = 0.12;

	brsstrcpy(&gDests[DEST_PIPETTE_2].Entry.Name,&"Pipette 2 Entry");
	gDests[DEST_PIPETTE_2].Entry.PathPoints[0].X = 0.42;
	gDests[DEST_PIPETTE_2].Entry.PathPoints[0].Y = 0.12;
	gDests[DEST_PIPETTE_2].Entry.Length = 1;

	brsstrcpy(&gDests[DEST_PIPETTE_2].Exit.Name,&"Pipette 2 Exit");
	gDests[DEST_PIPETTE_2].Exit.PathPoints[0].X = 0.30;
	gDests[DEST_PIPETTE_2].Exit.PathPoints[0].Y = 0.12;
	gDests[DEST_PIPETTE_2].Exit.Length = 1;

	//******Tips Destination
	brsstrcpy(&gDests[DEST_TIPS].StationName,&"Tips");
	gDests[DEST_TIPS].Position.X = 0.66;
	gDests[DEST_TIPS].Position.Y = 0.30;
	gDests[DEST_TIPS].RecoveryPts.X = 0.66;
	gDests[DEST_TIPS].RecoveryPts.Y = 0.30;

	brsstrcpy(&gDests[DEST_TIPS].Entry.Name,&"Tips Entry");
	gDests[DEST_TIPS].Entry.PathPoints[0].X = 0.54;
	gDests[DEST_TIPS].Entry.PathPoints[0].Y = 0.42;
	gDests[DEST_TIPS].Entry.PathPoints[1].X = 0.54;
	gDests[DEST_TIPS].Entry.PathPoints[1].Y = 0.30;
	gDests[DEST_TIPS].Entry.Length = 2;

	brsstrcpy(&gDests[DEST_TIPS].Exit.Name,&"Tips Exit");
	gDests[DEST_TIPS].Exit.PathPoints[0].X = 0.54;
	gDests[DEST_TIPS].Exit.PathPoints[0].Y = 0.30;
	gDests[DEST_TIPS].Exit.Length = 1;

	//******Dye Destination
	brsstrcpy(&gDests[DEST_DYE].StationName,&"Dye");
	gDests[DEST_DYE].Position.X = 0.66;
	gDests[DEST_DYE].Position.Y = 0.42;
	gDests[DEST_DYE].RecoveryPts.X = 0.66;
	gDests[DEST_DYE].RecoveryPts.Y = 0.42;

	brsstrcpy(&gDests[DEST_DYE].Entry.Name,&"Dye Entry");
	gDests[DEST_DYE].Entry.PathPoints[0].X = 0.54;
	gDests[DEST_DYE].Entry.PathPoints[0].Y = 0.42;
	gDests[DEST_DYE].Entry.Length = 1;

	brsstrcpy(&gDests[DEST_DYE].Exit.Name,&"Dye Exit");
	gDests[DEST_DYE].Exit.PathPoints[0].X = 0.54;
	gDests[DEST_DYE].Exit.PathPoints[0].Y = 0.42;
	gDests[DEST_DYE].Exit.Length = 1;

	//Define the Waypoints

	//******** Way Point 1
	brsstrcpy(&gWps[WP_1].Name,&"Waypoint 1");
	gWps[WP_1].Position.X = 0.30;
	gWps[WP_1].Position.Y = 0.42;
	gWps[WP_1].NextWaypoint = WP_2;
	gWps[WP_1].Destinations[0] = DEST_PIPETTE_1;

	//******** Way Point 2
	brsstrcpy(&gWps[WP_2].Name,&"Waypoint 2");
	gWps[WP_2].Position.X = 0.42;
	gWps[WP_2].Position.Y = 0.42;
	gWps[WP_2].NextWaypoint = WP_3;
	gWps[WP_2].Destinations[0] = DEST_DYE;
	gWps[WP_2].Destinations[1] = DEST_TIPS;

	//******** Way Point 3
	brsstrcpy(&gWps[WP_3].Name,&"Waypoint 3");
	gWps[WP_3].Position.X = 0.42;
	gWps[WP_3].Position.Y = 0.30;
	gWps[WP_3].NextWaypoint = WP_4;
	gWps[WP_3].Destinations[0] = DEST_PIPETTE_2;

	//******** Way Point 4
	brsstrcpy(&gWps[WP_4].Name,&"Waypoint 4");
	gWps[WP_4].Position.X = 0.30;
	gWps[WP_4].Position.Y = 0.30;
	gWps[WP_4].NextWaypoint = WP_1;
	gWps[WP_4].Destinations[0] = DEST_ANALYZER;
	gWps[WP_4].Destinations[1] = DEST_INCUBATOR;

	//******** Way Point 5
	brsstrcpy(&gWps[WP_5].Name,&"Waypoint 5");
	gWps[WP_5].Position.X = 0.54;
	gWps[WP_5].Position.Y = 0.30;
	gWps[WP_5].NextWaypoint = WP_3;
}
```

### Program Logical/Source/Core/DyeTipStations (ANSIC)

#### Types.typ
```iecst
TYPE
	GenericStationStateEnum :
		(
		GEN_OFF,
		GEN_STARTUP,
		GEN_READY,
		GEN_WAIT_SHUTTLE,
		GEN_WAIT_REQUEST,
		GEN_ERROR
		);
END_TYPE
```

#### Variables.var
```iecst
VAR
	dyeStFb : stnGeneric;
	dyeState : GenericStationStateEnum;
	tipsStFb : stnGeneric;
	tipsState : GenericStationStateEnum;
END_VAR
```

#### Cyclic.c
```c
#include <bur/plctypes.h>

#ifdef _DEFAULT_INCLUDES
	#include <AsDefault.h>
#endif

#define TRUE 1
#define FALSE 0

/*

	General Station IF needs
		Cmd.Enable
		Cmd.Run

	//Incubator station
		When requested send the shuttle away to the requested destination

	//Analyzer
		When requested, empty the completed well plate, reload the fresh one
		Make decision on if you should send to Pipette 1, 2 or a garage station

	//Dye and Tips stations
		Controlled together as a garage
			Garage publishes current status of the garages and their types of shuttles (if present)
		You make a request to the garage to request a shuttle of type to send to provided destination
		When Shuttle is present: Publish the type of shuttle present
		when requested, send the shuttle to the requested station

	Shuttle User Data
		Destination
		RecipeId
		ShuttleType
			WellPlate
			CellSample
			Tips
			Dye
		WellPlate Wells Status[bool:96]

	Recipe Definition
		FillTime
		NumSamples
		[Sample]
			Sample: Color
			SampleCount: 1-x
*/

void _CYCLIC ProgramCyclic(void)
{
	gStationsIf.Sts.IncubatorActive = dyeStFb.Active;

	//Tips Station Logic
	switch (tipsState)
	{
		case GEN_OFF:
			if(gStationsIf.Cmd.Enable){
				tipsStFb.Destination = &gDests[DEST_TIPS].Destination;
				tipsStFb.Velocity = gSysRecipe.DefaultVel;
				tipsStFb.Accel = gSysRecipe.DefaultAccel;
				tipsStFb.WaitTime = 0;//gSysRecipe.DefaultWaitTime;
				tipsStFb.ShuttleType = SH_TIPS;
				tipsStFb.Enable = TRUE;

				tipsState = GEN_STARTUP;
			}
			break;
		case GEN_STARTUP:
			if(tipsStFb.Active){
				tipsState = GEN_READY;
			}
			break;
		case GEN_READY:
			if(gStationsIf.Cmd.Run){
				tipsStFb.Run = TRUE;

				tipsState = GEN_WAIT_REQUEST;
			}
			break;
		case GEN_WAIT_SHUTTLE:
			gStationsIf.Sts.TipsShuttlePresent = tipsStFb.ShuttlePresent;
			if(gStationsIf.Sts.TipsShuttlePresent){
				//gStationsIf.Cmd.RequestTip = FALSE;
				tipsState = GEN_WAIT_REQUEST;
			}

			break;
		case GEN_WAIT_REQUEST:
			gStationsIf.Sts.TipsShuttlePresent= tipsStFb.ShuttlePresent;
			if(gStationsIf.Cmd.RequestTip){
				tipsStFb.NextDestination = &gDests[gStationsIf.Par.Tip.RequestDestination].Destination;
				tipsStFb.Waypoint = &gWps[WP_5].Waypoint;
				tipsStFb.Send = TRUE;

				if(!tipsStFb.ShuttlePresent){
					tipsStFb.Send = FALSE;
					tipsState = GEN_WAIT_SHUTTLE;
				}
			}
			break;
	}

	//Dye Logic
	switch (dyeState)
	{
		case GEN_OFF:
			if(gStationsIf.Cmd.Enable){
				dyeStFb.Destination = &gDests[DEST_DYE].Destination;
				dyeStFb.Velocity = gSysRecipe.DefaultVel;
				dyeStFb.Accel = gSysRecipe.DefaultAccel;
				dyeStFb.WaitTime = 0;//gSysRecipe.DefaultWaitTime;
				dyeStFb.ShuttleType = SH_DYE;
				dyeStFb.Enable = TRUE;

				dyeState = GEN_STARTUP;
			}
			break;
		case GEN_STARTUP:
			if(dyeStFb.Active){
				dyeState = GEN_READY;
			}
			break;
		case GEN_READY:
			if(gStationsIf.Cmd.Run){
				dyeStFb.Run = TRUE;

				dyeState = GEN_WAIT_REQUEST;
			}
			break;
		case GEN_WAIT_SHUTTLE:
			gStationsIf.Sts.DyeShuttlePresent = dyeStFb.ShuttlePresent;
			if(gStationsIf.Sts.DyeShuttlePresent){
				dyeState = GEN_WAIT_REQUEST;
			}
			break;
		case GEN_WAIT_REQUEST:
			gStationsIf.Sts.DyeShuttlePresent  = dyeStFb.ShuttlePresent;
			//Adding the Request tip check to try and prevent a deadlock
			if(gStationsIf.Cmd.RequestDye && !gStationsIf.Cmd.RequestTip){
				dyeStFb.NextDestination = &gDests[gStationsIf.Par.Dye.RequestDestination].Destination;
				dyeStFb.Waypoint = &gWps[WP_5].Waypoint;
				dyeStFb.Send = TRUE;

				if(!dyeStFb.ShuttlePresent){
					dyeStFb.Send = FALSE;
					dyeState = GEN_WAIT_SHUTTLE;
				}
			}
			break;
	}
	stnGeneric(&dyeStFb);
	stnGeneric(&tipsStFb);
}
```

#### Init.c
```c
#include <bur/plctypes.h>

#ifdef _DEFAULT_INCLUDES
	#include <AsDefault.h>
#endif

void _INIT ProgramInit(void)
{

}
```

### Program Logical/Source/Core/Stations (ANSIC)

#### Types.typ
```iecst
TYPE
	IncubatorStationStateEnum :
		(
		INC_OFF,
		INC_STARTUP,
		INC_READY,
		INC_WAIT_SHUTTLE,
		INC_WAIT_REQUEST,
		INC_ERROR
		);
	AnalyzerStationStateEnum :
		(
		ANALYZER_OFF,
		ANALYZER_STARTUP,
		ANALYZER_READY,
		ANALYZER_WAIT_SHUTTLE,
		ANALYZER_WAIT_REQUEST,
		ANALYZER_REQUEST_SAMPLE,
		ANALYZER_WAIT_PIPETTE_READY,
		ANALYZER_ERROR
		);
END_TYPE
```

#### Variables.var
```iecst
VAR
	initChecked : BOOL;
	shCount : USINT;
	incubatorStFb : stnGeneric;
	incubatorState : IncubatorStationStateEnum;
	analyzerState : AnalyzerStationStateEnum;
	analyzerStFb : stnGeneric;
END_VAR
```

#### Cyclic.c
```c
#include <bur/plctypes.h>

#ifdef _DEFAULT_INCLUDES
#include <AsDefault.h>
#endif

#define TRUE 1
#define FALSE 0

/*

	General Station IF needs
		Cmd.Enable
		Cmd.Run

	//Incubator station
		When requested send the shuttle away to the requested destination

	//Analyzer
		When requested, empty the completed well plate, reload the fresh one
		Make decision on if you should send to Pipette 1, 2 or a garage station

	//Dye and Tips stations
		Controlled together as a garage
			Garage publishes current status of the garages and their types of shuttles (if present)
		You make a request to the garage to request a shuttle of type to send to provided destination
		When Shuttle is present: Publish the type of shuttle present
		when requested, send the shuttle to the requested station

	Shuttle User Data
		Destination
		RecipeId
		ShuttleType
			WellPlate
			CellSample
			Tips
			Dye
		WellPlate Wells Status[bool:96]

	Recipe Definition
		FillTime
		NumSamples
		[Sample]
			Sample: Color
			SampleCount: 1-x
*/

void _CYCLIC ProgramCyclic(void)
{
	gStationsIf.Sts.IncubatorActive = incubatorStFb.Active;

	//Incubator Logic
	switch (incubatorState)
	{
		case INC_OFF:
			if(gStationsIf.Cmd.Enable){
				incubatorStFb.Destination = &gDests[DEST_INCUBATOR].Destination;
				incubatorStFb.Velocity = gSysRecipe.DefaultVel;
				incubatorStFb.Accel = gSysRecipe.DefaultAccel;
				incubatorStFb.WaitTime = gSysRecipe.DefaultWaitTime * 2;
				incubatorStFb.ShuttleType = SH_SAMPLE;
				incubatorStFb.Enable = TRUE;

				incubatorState = INC_STARTUP;
			}
			break;
		case INC_STARTUP:
			if(incubatorStFb.Active){
				incubatorState = INC_READY;
			}
			break;
		case INC_READY:
			if(gStationsIf.Cmd.Run){
				incubatorStFb.Run = TRUE;

				incubatorState = INC_WAIT_SHUTTLE;
			}
			break;
		case INC_WAIT_SHUTTLE:
			gStationsIf.Sts.IncubatorShuttlePresent = incubatorStFb.ShuttlePresent;
			if(incubatorStFb.ShuttlePresent){
				gShIfs[2].Cfg.RouterShuttle = incubatorStFb.internal.fbs.destMonFb.RouterShuttle; //Hack to set the RouterSh interface
				//This is all an ugly hack
				incubatorStFb.ShUserData.CurrentColor = COLOR_UNDEF;
				rl6dShCopyUserDataSync(&incubatorStFb.internal.fbs.destMonFb.RouterShuttle,rl6dSH_COPY_USER_DATA_WRITE,&incubatorStFb.ShUserData,sizeof(UserDataType));

				//end hack
				incubatorState = INC_WAIT_REQUEST;
			}
			break;
		case INC_WAIT_REQUEST:
			gStationsIf.Sts.IncubatorShuttlePresent = incubatorStFb.ShuttlePresent;
			if(gStationsIf.Cmd.RequestIncubator){
				incubatorStFb.NextDestination = &gDests[gStationsIf.Par.Incubator.NextStation].Destination;
				incubatorStFb.Waypoint = &gWps[gStationsIf.Par.Incubator.Waypoint].Waypoint;
				incubatorStFb.ShColor = gStationsIf.Par.Incubator.SampleType;
				incubatorStFb.Send = TRUE;

				if(!incubatorStFb.ShuttlePresent){
					gStationsIf.Cmd.RequestIncubator = FALSE;
					incubatorStFb.Send = FALSE;
					incubatorState = INC_WAIT_SHUTTLE;
				}
			}
			break;
	}

	//Analyzer Logic
	switch (analyzerState)
	{
		case ANALYZER_OFF:
			if(gStationsIf.Cmd.Enable){
				analyzerStFb.Destination = &gDests[DEST_ANALYZER].Destination;
				gStationsIf.Par.Analyzer.Waypoint = WP_1;
				analyzerStFb.Velocity = gSysRecipe.DefaultVel;
				analyzerStFb.Accel = gSysRecipe.DefaultAccel;
				analyzerStFb.WaitTime = gSysRecipe.DefaultWaitTime;
				analyzerStFb.ShuttleType = SH_WELL;
				analyzerStFb.ResetData = TRUE;
				analyzerStFb.Enable = TRUE;

				analyzerState = ANALYZER_STARTUP;
			}
			break;
		case ANALYZER_STARTUP:
			if(analyzerStFb.Active){
				analyzerState = ANALYZER_READY;
			}
			break;
		case ANALYZER_READY:
			if(gStationsIf.Cmd.Run){
				analyzerStFb.Run = TRUE;

				analyzerState = ANALYZER_WAIT_SHUTTLE;
			}
			break;
		case ANALYZER_WAIT_SHUTTLE:
			gStationsIf.Sts.AnalyzerShuttlePresent = analyzerStFb.ShuttlePresent;
			if(analyzerStFb.ShuttlePresent){
				if(!initChecked){
					gShIfs[shCount].Cfg.RouterShuttle = analyzerStFb.internal.fbs.destMonFb.RouterShuttle;
					shCount++;
					if(shCount==2)
						initChecked = TRUE;
				}
				analyzerState = ANALYZER_WAIT_REQUEST;

			}
			break;
		case ANALYZER_WAIT_REQUEST:
			gStationsIf.Sts.AnalyzerShuttlePresent = analyzerStFb.ShuttlePresent;
			if(gStationsIf.Cmd.RequestAnalyzer){
				analyzerStFb.NextDestination = &gDests[gStationsIf.Par.Analyzer.NextStation].Destination;
				analyzerStFb.Waypoint = &gWps[gStationsIf.Par.Analyzer.Waypoint].Waypoint;
				analyzerState = ANALYZER_WAIT_PIPETTE_READY;
			}

			if(analyzerStFb.ShuttlePresent && (gStationsIf.Sts.PipetteReadyForShuttle[0] || gStationsIf.Sts.PipetteReadyForShuttle[1])){
				//if we have a shuttle and either pipette station is ready, we should send a sample to it
				analyzerState = ANALYZER_REQUEST_SAMPLE;
			}

			break;
		case ANALYZER_REQUEST_SAMPLE:
			if(!gStationsIf.Cmd.RequestIncubator){
				gStationsIf.Cmd.RequestIncubator = TRUE;

				if(gStationsIf.Sts.PipetteReadyForShuttle[0]){
					//This is all an ugly hack
					analyzerStFb.ShUserData.Recipe = gSysRecipe.WellRecipe[0];
					rl6dShCopyUserDataSync(&analyzerStFb.internal.fbs.destMonFb.RouterShuttle,rl6dSH_COPY_USER_DATA_WRITE,&analyzerStFb.ShUserData,sizeof(UserDataType));
					gStationsIf.Par.Incubator.SampleType = analyzerStFb.ShUserData.Recipe.Samples[0].Sample;
					//end hack
					gStationsIf.Par.Incubator.NextStation = DEST_PIPETTE_1;
					gStationsIf.Sts.PipetteReadyForShuttle[0] = FALSE;
				}
				else if (gStationsIf.Sts.PipetteReadyForShuttle[1]){
					//This is all an ugly hack
					analyzerStFb.ShUserData.Recipe = gSysRecipe.WellRecipe[1];
					rl6dShCopyUserDataSync(&analyzerStFb.internal.fbs.destMonFb.RouterShuttle,rl6dSH_COPY_USER_DATA_WRITE,&analyzerStFb.ShUserData,sizeof(UserDataType));
					gStationsIf.Par.Incubator.SampleType = analyzerStFb.ShUserData.Recipe.Samples[0].Sample;
					//end hack

					gStationsIf.Par.Incubator.NextStation = DEST_PIPETTE_2;
					gStationsIf.Sts.PipetteReadyForShuttle[1] = FALSE;
				}
				analyzerState = ANALYZER_WAIT_REQUEST;
			}
			break;
		case ANALYZER_WAIT_PIPETTE_READY:
			gStationsIf.Sts.AnalyzerShuttlePresent = analyzerStFb.ShuttlePresent;

			analyzerStFb.Recipe = gSysRecipe.WellRecipe[gStationsIf.Par.Analyzer.NextStation - DEST_PIPETTE_1];
			analyzerStFb.ApplyRecipe = TRUE;
			analyzerStFb.Send = TRUE;
			if(!analyzerStFb.ShuttlePresent){
				gStationsIf.Cmd.RequestAnalyzer = FALSE;
				analyzerStFb.Send = FALSE;
				analyzerState = ANALYZER_WAIT_SHUTTLE;
			}

			break;
	}
	stnGeneric(&incubatorStFb);
	stnGeneric(&analyzerStFb);
}
```

#### Init.c
```c
#include <bur/plctypes.h>

#ifdef _DEFAULT_INCLUDES
	#include <AsDefault.h>
#endif

void _INIT ProgramInit(void)
{
	vel = 0.25;
	accel = 5;
}
```

### Program Logical/Source/Core/PipetteStations (ANSIC)

#### Types.typ
```iecst
TYPE
	PipetteStationStateEnum :
		(
		PIP_OFF,
		PIP_STARTUP,
		PIP_READY,
		PIP_REQUEST_TIP,
		PIP_CHANGE_TIP,
		PIP_REQUEST_SAMPLE,
		PIP_WAIT_SAMPLE,
		PIP_OPERATE_SAMPLE,
		PIP_REQUEST_SHUTTLE,
		PIP_WAIT_WELL_TO_ARRIVE,
		PIP_PROCESS_SHUTTLE,
		PIP_REQUEST_DYE,
		PIP_PROCESS_DYE,
		PIP_CHECK_RECIPE,
		PIP_SEND_ANALYZER,
		PIP_ERROR
		);
	PipetteIfTyp : 	STRUCT
		TipNeedReplace : BOOL;
		DyePresent : BOOL;
		SamplePresent : BOOL;
		shuttleIf : rl6dShuttleType;
		ShuttleOperating : BOOL;
		CurrentSample : ColorEnum;
		NextSample : ColorEnum;
		PipettePosition : REAL;
	END_STRUCT;
END_TYPE
```

#### Variables.var
```iecst
VAR
	i : USINT;
	pipetteState : ARRAY[0..1] OF PipetteStationStateEnum;
	pipetteFb : ARRAY[0..1] OF stnPipette;
	shIf : ARRAY[0..1] OF PipetteIfTyp;
	shMoveFb : ARRAY[0..1] OF rl6dShuttleMoveDestination;
END_VAR
```

#### Cyclic.c
```c
#include <bur/plctypes.h>

#ifdef _DEFAULT_INCLUDES
	#include <AsDefault.h>
#endif

#define TRUE 1
#define FALSE 0

/*
		//Pipette 1/2
		when a shuttle arrives
			Tips or Dye
				Wait for a set amount of time
				if pipette 1/2 Tips/Dye is needed > Send to Pipette 1/2
				else > send to tips/dye
			Well plate
				move shuttle to X/Y position corresponding to recipe (grid based position)
				wait Defined time
				go to next recipe index
				repeat until sample set completed
				if recipeIsDone
					sendToAnalyzer
				else:
					request Tip
				When Tip request has been answered
					send shuttle to tip station

		The TBD destinations are something passed into the station where to send it? Maybe defined by a global recipe?
*/

/*
	Wait for a shuttle to get assigned
		That shuttle defines the recipe we'll be using
		When tip enroute, if shuttle is at pipette, send shuttle to none
		When tip arrives, wait time to complete, request sample from incubator, Send Tip to tip destination
		when sample arrives, wait time to complete, send sample back to incubator, Update shuttle to go to Pipette
		When well plate arrives, wait for process to complete (should be doing indexing filling at that point)
		when process completed, request Tip, send shuttle to none
		When tip arrives, wait time to complete, send tip back to tips, request dye
		when dye completes, send back to dye station, update shuttle to go back to Pipette
		when sample arrives, doing the same waiting for indexing again

		at this point, we've completed a sample set, so increment the sample set.
		if recpipe is finished, send to analyzer and head back to 1st wait state
		otherwise, repeat process again (request new tip etc)

*/
void _CYCLIC ProgramCyclic(void)
{

	for(i = 0; i < 2; i++){

		//Pipette Logic
		switch (pipetteState[i])
		{
			case PIP_OFF:
				if(gStationsIf.Cmd.Enable){
					pipetteFb[i].Velocity = gSysRecipe.DefaultVel;
					pipetteFb[i].Accel = gSysRecipe.DefaultAccel;
					pipetteFb[i].WaitTime = gSysRecipe.DefaultWaitTime;
					pipetteFb[i].InitialId = i;
					pipetteFb[i].Enable = TRUE;

					pipetteState[i] = PIP_STARTUP;
				}
				break;

			case PIP_STARTUP:
				if(pipetteFb[i].Active){
					gStationsIf.Sts.PipetteActive[i] = TRUE;
					shIf[i].PipettePosition = gSysRecipe.PipettePars.HomePosition;
					pipetteState[i] = PIP_READY;
				}
				break;
			case PIP_READY:
				pipetteState[i] = PIP_REQUEST_TIP;

				break;
			case PIP_REQUEST_TIP:
				//Waiting for a shuttle to arrive that is of type tip
				if(!gStationsIf.Cmd.RequestTip){
					gStationsIf.Cmd.RequestTip = 1;
					gStationsIf.Par.Tip.RequestDestination = DEST_PIPETTE_1 + i;
				}
				if(pipetteFb[i].ShuttlePresent && pipetteFb[i].ShUserData.ShType == SH_TIPS){
					gStationsIf.Cmd.RequestTip = FALSE;
					pipetteState[i] = PIP_CHANGE_TIP;
				}
				break;
			case PIP_CHANGE_TIP:
				if(pipetteFb[i].WaitComplete){
					shIf[i].TipNeedReplace = FALSE;
					shIf[i].CurrentSample = COLOR_GRAY;
					pipetteFb[i].NextDestination = &gDests[DEST_TIPS].Destination;
					pipetteFb[i].Send = TRUE;
					if(!shIf[i].ShuttleOperating){
						//We haven't received a shuttle yet, we should go ahead and tell the system we're ready to receive a sample and shuttle and wait for one.
						gStationsIf.Sts.PipetteReadyForShuttle[i] = TRUE;
						pipetteState[i] = PIP_WAIT_SAMPLE;
					}
					else{
						if(!shIf[i].SamplePresent){
							pipetteState[i] = PIP_REQUEST_SAMPLE;
						}
						else{
							pipetteState[i] = PIP_REQUEST_DYE;
						}
					}
				}
				break;

			case PIP_REQUEST_SAMPLE:
				if(!gStationsIf.Cmd.RequestIncubator){
					gStationsIf.Cmd.RequestIncubator = TRUE;
					gStationsIf.Par.Incubator.SampleType = shIf[i].NextSample;
					gStationsIf.Par.Incubator.NextStation = DEST_PIPETTE_1 + i;
					pipetteState[i] = PIP_WAIT_SAMPLE;
				}
				break;
			case PIP_WAIT_SAMPLE:
				if(pipetteFb[i].ShuttlePresent && pipetteFb[i].ShUserData.ShType == SH_SAMPLE){
					pipetteState[i] = PIP_OPERATE_SAMPLE;
				}
				break;
			case PIP_OPERATE_SAMPLE:
				if(pipetteFb[i].WaitComplete){
					shIf[i].CurrentSample = pipetteFb[i].ShUserData.CurrentColor;
					pipetteFb[i].NextDestination = &gDests[DEST_INCUBATOR].Destination;
					pipetteFb[i].Send = TRUE;

					pipetteFb[i].DyePresent = FALSE;

					pipetteState[i] = PIP_REQUEST_SHUTTLE;
				}
				break;
			case PIP_REQUEST_SHUTTLE:
				if(!gStationsIf.Cmd.RequestAnalyzer && !shIf[i].ShuttleOperating){
					gStationsIf.Cmd.RequestAnalyzer = TRUE;
					gStationsIf.Par.Analyzer.NextStation = DEST_PIPETTE_1 + i;
					shIf[i].ShuttleOperating = TRUE;

					pipetteState[i] = PIP_WAIT_WELL_TO_ARRIVE;
				}
				else if(shIf[i].ShuttleOperating){
					//Shuttle is already present, so we need to request it from the shMove block
					shMoveFb[i].Destination = &gDests[DEST_PIPETTE_1 + i].Destination;
					shMoveFb[i].Velocity = gSysRecipe.DefaultVel;
					shMoveFb[i].Acceleration = gSysRecipe.DefaultAccel;
					shMoveFb[i].RouterShuttle = &shIf[i].shuttleIf;
					shMoveFb[i].Execute = TRUE;

					pipetteState[i] = PIP_WAIT_WELL_TO_ARRIVE;
				}

				break;
			case PIP_WAIT_WELL_TO_ARRIVE:
				if(pipetteFb[i].ShuttlePresent && pipetteFb[i].ShUserData.ShType == SH_WELL){
					shMoveFb[i].Execute = FALSE;

					gStationsIf.Cmd.RequestPipette[i] = FALSE;
					pipetteState[i] = PIP_PROCESS_SHUTTLE;
				}
				break;
			case PIP_PROCESS_SHUTTLE:
				if(pipetteFb[i].OperateDone){
					if(!shIf[i].SamplePresent){
						shIf[i].shuttleIf = pipetteFb[i].Shuttle;
						shIf[i].SamplePresent = TRUE;
						shIf[i].TipNeedReplace = TRUE;
						pipetteFb[i].NextDestination = &gDests[DEST_DEFAULT].Destination;
						pipetteFb[i].Send = TRUE;

						pipetteState[i] = PIP_REQUEST_TIP;
					}
					else{
						//Need to go check on the recipe now
						pipetteState[i] = PIP_CHECK_RECIPE;
					}
				}
				break;
			case PIP_REQUEST_DYE:
				if(!gStationsIf.Cmd.RequestDye){
					gStationsIf.Cmd.RequestDye = TRUE;
					gStationsIf.Par.Dye.RequestDestination = DEST_PIPETTE_1 + i;
				}
				if(pipetteFb[i].ShuttlePresent && pipetteFb[i].ShUserData.ShType == SH_DYE){
					gStationsIf.Cmd.RequestDye = FALSE;
					pipetteState[i] = PIP_PROCESS_DYE;
				}
				break;
			case PIP_PROCESS_DYE:
				if(pipetteFb[i].WaitComplete){
					shIf[i].DyePresent = TRUE;
					pipetteFb[i].NextDestination = &gDests[DEST_DYE].Destination;
					pipetteFb[i].Send = TRUE;
					shIf[i].CurrentSample = COLOR_WHITE;
					pipetteFb[i].DyePresent = TRUE;

					if(shIf[i].SamplePresent){
						shMoveFb[i].Destination = &gDests[DEST_PIPETTE_1 + i].Destination;
						shMoveFb[i].Velocity = gSysRecipe.DefaultVel;
						shMoveFb[i].Acceleration = gSysRecipe.DefaultAccel;
						shMoveFb[i].RouterShuttle = &shIf[i].shuttleIf;
						shMoveFb[i].Execute = TRUE;

						pipetteState[i] = PIP_WAIT_WELL_TO_ARRIVE;
					}
					else{
						pipetteState[i] = PIP_REQUEST_SHUTTLE;
					}
				}
				break;
			case PIP_CHECK_RECIPE:
				//If the sample and well count == numRows * numColumns, then we're done
					//Send the shuttle to the analyzer, and reset any flags to start the process over again
				//Otherwise, request the next sample and keep going on
				if(pipetteFb[i].ShUserData.Recipe.SampleWellCount == (pipetteFb[i].WellPlateInfo.NumColumns * pipetteFb[i].WellPlateInfo.NumRows) &&
						pipetteFb[i].ShUserData.Recipe.DyeWellCount == (pipetteFb[i].WellPlateInfo.NumColumns * pipetteFb[i].WellPlateInfo.NumRows)){
					shIf[i].DyePresent = FALSE;
					shIf[i].SamplePresent = FALSE;
					pipetteFb[i].DyePresent = FALSE;
					shIf[i].TipNeedReplace = FALSE;
					brsmemset(&shIf[i].shuttleIf,0,sizeof(shIf[i].shuttleIf));
					pipetteFb[i].NextDestination = &gDests[DEST_ANALYZER].Destination;
					pipetteFb[i].Send = TRUE;
					shIf[i].ShuttleOperating = FALSE;

					pipetteState[i] = PIP_SEND_ANALYZER;
				}
				else{
					shIf[i].DyePresent = FALSE;
					shIf[i].shuttleIf = pipetteFb[i].Shuttle;
					shIf[i].SamplePresent = FALSE;
					shIf[i].TipNeedReplace = TRUE;
					pipetteFb[i].NextDestination = &gDests[DEST_DEFAULT].Destination;
					pipetteFb[i].Send = TRUE;
					pipetteFb[i].DyePresent = FALSE;
					shIf[i].NextSample = pipetteFb[i].ShUserData.Recipe.Samples[pipetteFb[i].ShUserData.Recipe.CurrentSample].Sample;
					pipetteState[i] = PIP_REQUEST_TIP;
				}
				break;
			case PIP_SEND_ANALYZER:
				if(!pipetteFb[i].ShuttlePresent){
					pipetteFb[i].Send = FALSE;
					pipetteState[i] = PIP_REQUEST_TIP;
				}
				break;
		}
		stnPipette(&pipetteFb[i]);
		rl6dShuttleMoveDestination(&shMoveFb[i]);
		if(pipetteFb[i].Send && !pipetteFb[i].ShuttlePresent){
			pipetteFb[i].Send = FALSE;
		}
		if(shMoveFb[i].Active && shMoveFb[i].Execute){
			shMoveFb[i].Execute = FALSE;
		}
	}
}
```

#### Init.c
```c
#include <bur/plctypes.h>

#ifdef _DEFAULT_INCLUDES
	#include <AsDefault.h>
#endif

void _INIT ProgramInit(void)
{
	pipetteFb[0].Destination = &gDests[DEST_PIPETTE_1].Destination;
	pipetteFb[0].Waypoint = &gWps[WP_2].Waypoint;
	pipetteFb[0].FirstDestination = &gDests[DEST_ANALYZER].Destination;

	pipetteFb[1].Destination = &gDests[DEST_PIPETTE_2].Destination;
	pipetteFb[1].Waypoint = &gWps[WP_4].Waypoint;
	pipetteFb[1].FirstDestination = &gDests[DEST_INCUBATOR].Destination;

	pipetteFb[0].WellPlateInfo.ColumnGap = 0.02;
	pipetteFb[0].WellPlateInfo.RowGap = 0.02;
	pipetteFb[0].WellPlateInfo.NumColumns = 4;
	pipetteFb[0].WellPlateInfo.NumRows = 4;
	pipetteFb[0].WellPlateInfo.OffsetX = 0.031;
	pipetteFb[0].WellPlateInfo.OffsetY = 0.031;

	pipetteFb[1].WellPlateInfo.ColumnGap = 0.02;
	pipetteFb[1].WellPlateInfo.RowGap = 0.02;
	pipetteFb[1].WellPlateInfo.NumColumns = 4;
	pipetteFb[1].WellPlateInfo.NumRows = 4;
	pipetteFb[1].WellPlateInfo.OffsetX = 0.031;
	pipetteFb[1].WellPlateInfo.OffsetY = 0.031;

	gSysRecipe.WellRecipe[0].CurrentSample = 0;
	gSysRecipe.WellRecipe[0].NumberSamples = 3;
	gSysRecipe.WellRecipe[0].Samples[0].CurrentCount = 0;
	gSysRecipe.WellRecipe[0].Samples[0].Sample = COLOR_DARK_BLUE;
	gSysRecipe.WellRecipe[0].Samples[0].SampleCount = 6;
	gSysRecipe.WellRecipe[0].Samples[1].CurrentCount = 0;
	gSysRecipe.WellRecipe[0].Samples[1].Sample = COLOR_DARK_GREEN;
	gSysRecipe.WellRecipe[0].Samples[1].SampleCount = 6;
	gSysRecipe.WellRecipe[0].Samples[2].CurrentCount = 0;
	gSysRecipe.WellRecipe[0].Samples[2].Sample = COLOR_DARK_YELLOW;
	gSysRecipe.WellRecipe[0].Samples[2].SampleCount = 4;

	gSysRecipe.WellRecipe[1].CurrentSample = 0;
	gSysRecipe.WellRecipe[1].NumberSamples = 4;
	gSysRecipe.WellRecipe[1].Samples[0].CurrentCount = 0;
	gSysRecipe.WellRecipe[1].Samples[0].Sample = COLOR_DARK_YELLOW;
	gSysRecipe.WellRecipe[1].Samples[0].SampleCount = 3;
	gSysRecipe.WellRecipe[1].Samples[1].CurrentCount = 0;
	gSysRecipe.WellRecipe[1].Samples[1].Sample = COLOR_DARK_BLUE;
	gSysRecipe.WellRecipe[1].Samples[1].SampleCount = 6;
	gSysRecipe.WellRecipe[1].Samples[2].CurrentCount = 0;
	gSysRecipe.WellRecipe[1].Samples[2].Sample = COLOR_RED;
	gSysRecipe.WellRecipe[1].Samples[2].SampleCount = 4;
	gSysRecipe.WellRecipe[1].Samples[3].CurrentCount = 0;
	gSysRecipe.WellRecipe[1].Samples[3].Sample = COLOR_DARK_GREEN;
	gSysRecipe.WellRecipe[1].Samples[3].SampleCount = 3;
}
```

### Library Logical/Source/Core/StnLogic (ANSIC)
Depends on: Router6D, standard, AsBrStr

#### Types.typ - Exported data types
```iecst
TYPE
	DestinationsEnum :
		(
		DEST_DEFAULT,
		DEST_INCUBATOR,
		DEST_ANALYZER,
		DEST_PIPETTE_1,
		DEST_PIPETTE_2,
		DEST_TIPS,
		DEST_DYE
		);
	ShuttleType :
		(
		SH_EMPTY,
		SH_WELL,
		SH_SAMPLE,
		SH_DYE,
		SH_TIPS
		);
	UserDataType : 	STRUCT
		shId : USINT;
		ShType : ShuttleType;
		CurrentColor : ColorEnum;
		Recipe : FillRecipeTyp;
		Wells : ARRAY[0..17]OF WellTyp;
	END_STRUCT;
	WellTyp : 	STRUCT
		Present : BOOL;
		Color : ColorEnum;
	END_STRUCT;
	ColorEnum :
		(
		COLOR_UNDEF,
		COLOR_BLACK,
		COLOR_RED,
		COLOR_PINK,
		COLOR_DARK_BLUE,
		COLOR_LIGHT_BLUE,
		COLOR_DARK_GREEN,
		COLOR_LIGHT_GREEN,
		COLOR_DARK_YELLOW,
		COLOR_LIGHT_YELLOW,
		COLOR_GRAY,
		COLOR_WHITE,
		COLOR_DARK_PURPLE,
		COLOR_LIGHT_PURPLE,
		COLOR_DARK_ORANGE,
		COLOR_LIGHT_ORANGE
		);
END_TYPE

(*Fill Recipe Types*)

TYPE
	FillRecipeTyp : 	STRUCT
		NumberSamples : USINT;
		CurrentSample : USINT;
		SampleWellCount : USINT;
		DyeWellCount : USINT;
		Samples : ARRAY[0..4]OF FillSampleTyp;
	END_STRUCT;
	FillSampleTyp : 	STRUCT
		Sample : ColorEnum;
		SampleCount : USINT;
		CurrentCount : USINT;
	END_STRUCT;
	WellPlateInfoTyp : 	STRUCT
		NumRows : USINT;
		NumColumns : USINT;
		RowGap : REAL;
		ColumnGap : REAL;
		OffsetX : REAL;
		OffsetY : REAL;
	END_STRUCT;
END_TYPE

(*Generic Station Types*)

TYPE
	stnGenericIntTyp : 	STRUCT
		state : stnGenericEnumTyp;
		errorState : stnGenericEnumTyp;
		fbs : stnGenericFbTyp;
	END_STRUCT;
	stnGenericEnumTyp :
		(
		STN_GENERIC_OFF,
		STN_GENERIC_INIT,
		STN_GENERIC_READY,
		STN_GENERIC_PROCESS,
		STN_GENERIC_WAIT_FOR_CMD,
		STN_GENERIC_SEND,
		STN_GENERIC_DONE,
		STN_GENERIC_ERROR,
		STN_GENERIC_RESET
		);
	stnGenericFbTyp : 	STRUCT
		destMonFb : rl6dDestinationMonitor;
		moveDestFb : rl6dShuttleMoveDestination;
		waitFb : TON;
	END_STRUCT;
END_TYPE

(*Pipette Station Types*)

TYPE
	stnPipetteIntTyp : 	STRUCT
		state : stnPipetteEnum;
		errorState : stnPipetteEnum;
		fillState : stnPipetteFillStatesEnum;
		fillPos : stnPipetteFillGridPosTyp;
		fbs : stnPipetteFbsTyp;
	END_STRUCT;
	stnPipetteEnum :
		(
		STN_PIPETTE_OFF,
		STN_PIPETTE_INIT,
		STN_PIPETTE_WAIT_FIRST,
		STN_PIPETTE_SEND_FIRST,
		STN_PIPETTE_READY,
		STN_PIPETTE_DO_WAIT,
		STN_PIPETTE_PROCESS,
		STN_PIPETTE_WAIT_FOR_CMD,
		STN_PIPETTE_SEND,
		STN_PIPETTE_DONE,
		STN_PIPETTE_ERROR,
		STN_PIPETTE_RESET
		);
	stnPipetteFbsTyp : 	STRUCT
		destMonFb : rl6dDestinationMonitor;
		moveDestFb : rl6dShuttleMoveDestination;
		waitFb : TON;
		moveInPlaneFb : MC_BR_MoveInPlane_Acp6D;
		moveArcFb : MC_BR_MoveArc_Acp6D;
	END_STRUCT;
	stnPipetteFillStatesEnum :
		(
		FILL_MOVE,
		FILL_FILL,
		FILL_SWIRL,
		FILL_CHECK_RECIPE
		);
	stnPipetteFillGridPosTyp : 	STRUCT
		X : USINT;
		Y : USINT;
	END_STRUCT;
END_TYPE
```

#### StnLogic.fun - Exported functions and function blocks
```iecst
{REDUND_ERROR} FUNCTION_BLOCK stnPipette (*TODO: Add your comment here*) (*$GROUP=User,$CAT=User,$GROUPICON=User.png,$CATICON=User.png*)
	VAR_INPUT
		Destination : REFERENCE TO rl6dDestinationType;
		InitialId : USINT;
		FirstDestination : REFERENCE TO rl6dDestinationType;
		Enable : BOOL;
		Operate : BOOL;
		Run : BOOL;
		Send : BOOL;
		NextDestination : REFERENCE TO rl6dDestinationType;
		Waypoint : REFERENCE TO rl6dWaypointType;
		WellPlateInfo : WellPlateInfoTyp;
		Velocity : REAL;
		Accel : REAL;
		DyePresent : BOOL;
		WaitTime : UDINT;
	END_VAR
	VAR_OUTPUT
		Active : BOOL;
		Error : BOOL;
		ErrorID : DINT;
		ShuttlePresent : BOOL;
		ShUserData : UserDataType;
		Shuttle : rl6dShuttleType;
		OperateDone : USINT;
		WaitComplete : BOOL;
	END_VAR
	VAR
		internal : stnPipetteIntTyp;
	END_VAR
END_FUNCTION_BLOCK

{REDUND_ERROR} FUNCTION_BLOCK stnGeneric (*TODO: Add your comment here*) (*$GROUP=User,$CAT=User,$GROUPICON=User.png,$CATICON=User.png*)
	VAR_INPUT
		Destination : REFERENCE TO rl6dDestinationType;
		Enable : BOOL;
		Run : BOOL;
		Send : BOOL;
		ResetData : BOOL;
		ShuttleType : ShuttleType;
		Recipe : FillRecipeTyp;
		ShColor : ColorEnum;
		ApplyRecipe : BOOL;
		NextDestination : REFERENCE TO rl6dDestinationType;
		Waypoint : REFERENCE TO rl6dWaypointType;
		Velocity : REAL;
		Accel : REAL;
		WaitTime : DINT;
	END_VAR
	VAR_OUTPUT
		Active : BOOL;
		Error : BOOL;
		ErrorID : UDINT;
		ShuttlePresent : BOOL;
		ShUserData : UserDataType;
		WaitComplete : BOOL;
	END_VAR
	VAR
		internal : stnGenericIntTyp;
	END_VAR
END_FUNCTION_BLOCK
```

#### stnGeneric.c
```c
#include <bur/plctypes.h>
#ifdef __cplusplus
	extern "C"
	{
#endif
#include "StnLogic.h"
#ifdef __cplusplus
	};
#endif

#define TRUE 1
#define FALSE 0

/* TODO: Add your comment here */
void stnGeneric(struct stnGeneric* fb)
{
	switch (fb->internal.state)
	{
		//******************** Off State
		case STN_GENERIC_OFF:
			if(fb->Enable){
				fb->internal.fbs.destMonFb.Destination = fb->Destination;
				fb->internal.fbs.destMonFb.Enable = TRUE;
				fb->internal.state = STN_GENERIC_INIT;
			}
			break;
		//******************** Initalize State
		case STN_GENERIC_INIT:

			if(fb->internal.fbs.destMonFb.Valid){
				fb->Active = TRUE;
			}

			if(fb->internal.fbs.destMonFb.Valid && fb->Run){
				fb->internal.state = STN_GENERIC_READY;
			}

			break;
		//******************** Ready and Waiting For a Shuttle State
		case STN_GENERIC_READY:
			if(fb->internal.fbs.destMonFb.ShuttlePresent){
				fb->ShuttlePresent = TRUE;
				fb->internal.fbs.waitFb.PT = fb->WaitTime;
				fb->internal.fbs.waitFb.IN = TRUE;
				rl6dShCopyUserDataSync(&fb->internal.fbs.destMonFb.RouterShuttle,rl6dSH_COPY_USER_DATA_READ,&fb->ShUserData,sizeof(fb->ShUserData));

				fb->internal.state = STN_GENERIC_PROCESS;
			}
			break;
		//******************** Processing State
		case STN_GENERIC_PROCESS:
			rl6dShCopyUserDataSync(&fb->internal.fbs.destMonFb.RouterShuttle,rl6dSH_COPY_USER_DATA_READ,&fb->ShUserData,sizeof(fb->ShUserData));
			if(fb->internal.fbs.waitFb.Q){
				fb->internal.fbs.waitFb.IN = FALSE;
				fb->WaitComplete = TRUE;

				fb->internal.state = STN_GENERIC_WAIT_FOR_CMD;
			}

			break;
		//******************** Waiting for the send command State
		case STN_GENERIC_WAIT_FOR_CMD:
			rl6dShCopyUserDataSync(&fb->internal.fbs.destMonFb.RouterShuttle,rl6dSH_COPY_USER_DATA_READ,&fb->ShUserData,sizeof(fb->ShUserData));
			if(fb->Send){
				//Update the user data
				if(fb->ResetData){
					brsmemset(&fb->ShUserData,0,sizeof(fb->ShUserData));
					fb->ErrorID = rl6dShCopyUserDataSync(&fb->internal.fbs.destMonFb.RouterShuttle,rl6dSH_COPY_USER_DATA_WRITE,&fb->ShUserData,sizeof(fb->ShUserData));
				}
				if(fb->ApplyRecipe){
					fb->ShUserData.Recipe = fb->Recipe;
				}
				fb->ShUserData.CurrentColor = fb->ShColor;
				fb->ShUserData.ShType = fb->ShuttleType;
				fb->ErrorID = rl6dShCopyUserDataSync(&fb->internal.fbs.destMonFb.RouterShuttle,rl6dSH_COPY_USER_DATA_WRITE,&fb->ShUserData,sizeof(fb->ShUserData));

				fb->internal.fbs.moveDestFb.RouterShuttle = &fb->internal.fbs.destMonFb.RouterShuttle;
				fb->internal.fbs.moveDestFb.Destination = fb->NextDestination;
				fb->internal.fbs.moveDestFb.Waypoint = fb->Waypoint;
				fb->internal.fbs.moveDestFb.Velocity = fb->Velocity;
				fb->internal.fbs.moveDestFb.Acceleration = fb->Accel;
				fb->internal.fbs.moveDestFb.Execute = TRUE;

				fb->internal.state = STN_GENERIC_SEND;
			}
			break;
		//******************** Send Shuttle State State
		case STN_GENERIC_SEND:
			if(fb->internal.fbs.moveDestFb.Error){
				fb->internal.errorState = fb->internal.state;
				fb->Error = TRUE;
				fb->ErrorID = fb->internal.fbs.moveDestFb.ErrorID;
				fb->internal.state = STN_GENERIC_ERROR;
			}
			else if(fb->internal.fbs.moveDestFb.Active){
				fb->internal.fbs.destMonFb.AcknowledgeShuttle = TRUE;
				if(!fb->internal.fbs.destMonFb.ShuttlePresent){
					fb->internal.fbs.destMonFb.AcknowledgeShuttle = FALSE;
					fb->internal.fbs.moveDestFb.Execute = FALSE;
					fb->ShuttlePresent = FALSE;
					fb->WaitComplete = FALSE;
					brsmemset(&fb->ShUserData,0,sizeof(fb->ShUserData));

					fb->internal.state = STN_GENERIC_DONE;
				}
			}
			break;
		//******************** Waiting for the Send Cmd To Drop State
		case STN_GENERIC_DONE:
			if(!fb->Send){
				fb->internal.state = STN_GENERIC_READY;
			}
			break;
		//******************** Error State
		case STN_GENERIC_ERROR:
			if(!fb->Enable){

			}
			break;
		//******************** Reset State
		case STN_GENERIC_RESET:

			break;
	}

	TON(&fb->internal.fbs.waitFb);
	rl6dDestinationMonitor(&fb->internal.fbs.destMonFb);
	rl6dShuttleMoveDestination(&fb->internal.fbs.moveDestFb);
}
```

#### stnPipette.c
```c
#include <bur/plctypes.h>
#ifdef __cplusplus
	extern "C"
	{
#endif
#include "StnLogic.h"
#ifdef __cplusplus
	};
#endif

#define TRUE 1
#define FALSE 0

/* TODO: Add your comment here */
void stnPipette(struct stnPipette* fb)
{
	switch (fb->internal.state)
	{
		//******************** Off State
		case STN_PIPETTE_OFF:
			if(fb->Enable){
				fb->internal.fbs.destMonFb.Destination = fb->Destination;
				fb->internal.fbs.destMonFb.Enable = TRUE;
				fb->internal.state = STN_PIPETTE_INIT;
			}
			break;
		//******************** Initalize State
		case STN_PIPETTE_INIT:

			if(fb->internal.fbs.destMonFb.Valid){
				fb->Active = TRUE;
				fb->internal.state = STN_PIPETTE_WAIT_FIRST;
			}
			break;
		//******************** Waiting For the First Shuttle States
		case STN_PIPETTE_WAIT_FIRST:
			if(fb->internal.fbs.destMonFb.ShuttlePresent){
				fb->internal.fbs.moveDestFb.RouterShuttle = &fb->internal.fbs.destMonFb.RouterShuttle;
				fb->internal.fbs.moveDestFb.Destination = fb->FirstDestination;
				fb->internal.fbs.moveDestFb.Waypoint = fb->Waypoint;
				fb->internal.fbs.moveDestFb.Velocity = fb->Velocity;
				fb->internal.fbs.moveDestFb.Acceleration = fb->Accel;
				fb->internal.fbs.moveDestFb.Execute = TRUE;

				fb->ShUserData.shId = fb->InitialId;
				rl6dShCopyUserDataSync(&fb->internal.fbs.destMonFb.RouterShuttle,rl6dSH_COPY_USER_DATA_WRITE,&fb->ShUserData,sizeof(fb->ShUserData));

				fb->internal.state = STN_PIPETTE_SEND_FIRST;
			}
			break;
		//******************** Sending the first shuttle state
		case STN_PIPETTE_SEND_FIRST:
			if(fb->internal.fbs.moveDestFb.Active){
				fb->internal.fbs.destMonFb.AcknowledgeShuttle = TRUE;
				if(!fb->internal.fbs.destMonFb.ShuttlePresent){
					fb->internal.fbs.moveDestFb.Execute = FALSE;
					fb->internal.fbs.destMonFb.AcknowledgeShuttle = FALSE;
					fb->internal.state = STN_PIPETTE_READY;
				}
			}
			break;
		//******************** Ready and Waiting For a Shuttle State
		case STN_PIPETTE_READY:
			fb->ShuttlePresent = fb->internal.fbs.destMonFb.ShuttlePresent;
			if(fb->internal.fbs.destMonFb.ShuttlePresent){
				fb->Shuttle = fb->internal.fbs.destMonFb.RouterShuttle;
				rl6dShCopyUserDataSync(&fb->internal.fbs.destMonFb.RouterShuttle,rl6dSH_COPY_USER_DATA_READ,&fb->ShUserData,sizeof(fb->ShUserData));
				if(fb->ShUserData.ShType != SH_WELL){
					fb->ShuttlePresent = TRUE;
					fb->internal.fbs.waitFb.PT = fb->WaitTime;
					fb->internal.fbs.waitFb.IN = TRUE;

					fb->internal.state = STN_PIPETTE_DO_WAIT;
				}
				else{
					USINT sampleIndex;
					sampleIndex = fb->ShUserData.Recipe.CurrentSample;
					fb->ShUserData.Recipe.Samples[sampleIndex].CurrentCount = 0;

					if(!fb->DyePresent){
						fb->internal.fillPos.Y = fb->ShUserData.Recipe.SampleWellCount / fb->WellPlateInfo.NumColumns;
						fb->internal.fillPos.X = fb->ShUserData.Recipe.SampleWellCount - (fb->internal.fillPos.Y * fb->WellPlateInfo.NumColumns);

					}
					else{
						fb->internal.fillPos.Y = fb->ShUserData.Recipe.DyeWellCount / fb->WellPlateInfo.NumColumns;
						fb->internal.fillPos.X = fb->ShUserData.Recipe.DyeWellCount - (fb->internal.fillPos.Y * fb->WellPlateInfo.NumColumns);
					}
					fb->internal.fbs.moveInPlaneFb.Shuttle = &fb->internal.fbs.destMonFb.Mc6DShuttle;
					fb->internal.fbs.moveInPlaneFb.Parameters.Velocity = fb->Velocity;
					fb->internal.fbs.moveInPlaneFb.Parameters.Acceleration = fb->Accel;
					fb->internal.fbs.moveInPlaneFb.Parameters.Path = mcACP6D_PATH_DIRECT;
					fb->internal.fbs.moveInPlaneFb.Parameters.Position.X = (fb->WellPlateInfo.OffsetX - fb->internal.fillPos.X * fb->WellPlateInfo.ColumnGap);
					fb->internal.fbs.moveInPlaneFb.Parameters.Position.Y = (fb->WellPlateInfo.OffsetY - fb->internal.fillPos.Y * fb->WellPlateInfo.RowGap);
					fb->internal.fbs.moveInPlaneFb.Parameters.Mode = mcACP6D_MOVE_RELATIVE;
					fb->internal.fbs.moveInPlaneFb.Execute = TRUE;

					fb->internal.fillState = FILL_MOVE;
					fb->internal.state = STN_PIPETTE_PROCESS;
				}
			}
			break;
		//******************** "Wait" process State
		case STN_PIPETTE_DO_WAIT:
			rl6dShCopyUserDataSync(&fb->internal.fbs.destMonFb.RouterShuttle,rl6dSH_COPY_USER_DATA_READ,&fb->ShUserData,sizeof(fb->ShUserData));
			if(fb->internal.fbs.waitFb.Q){
				fb->internal.fbs.waitFb.IN = FALSE;
				fb->WaitComplete = TRUE;

				fb->internal.state = STN_PIPETTE_WAIT_FOR_CMD;
			}

			break;
		//******************** Processing State
		case STN_PIPETTE_PROCESS:
			//in this state we're going to make the indexing movements around to fill up the shuttle with product

			switch (fb->internal.fillState)
			{
				case FILL_MOVE:
					if(fb->internal.fbs.moveInPlaneFb.Done){
						fb->internal.fbs.moveInPlaneFb.Execute = FALSE;

						fb->internal.fbs.waitFb.IN = TRUE;
						fb->internal.fbs.waitFb.PT = fb->WaitTime;

						fb->internal.fillState = FILL_FILL;
					}
					break;

				case FILL_FILL:
					if(fb->internal.fbs.waitFb.Q){
						fb->internal.fbs.waitFb.IN = FALSE;

						if(fb->DyePresent){
							fb->internal.fbs.moveArcFb.Shuttle = &fb->internal.fbs.destMonFb.Mc6DShuttle;
							fb->internal.fbs.moveArcFb.Parameters.Acceleration = 10.0;
							fb->internal.fbs.moveArcFb.Parameters.Velocity = 0.2;
							fb->internal.fbs.moveArcFb.Parameters.Angular.Center.X = -0.003;
							fb->internal.fbs.moveArcFb.Parameters.Angular.Center.Y = -0.003;
							fb->internal.fbs.moveArcFb.Parameters.Angular.Angle = 3.14*2*5;
							fb->internal.fbs.moveArcFb.Parameters.Mode = mcACP6D_MOVE_RELATIVE;
							fb->internal.fbs.moveArcFb.Parameters.Option = mcACP6D_ARC_ANGULAR;
							fb->internal.fbs.moveArcFb.Execute = TRUE;
							fb->internal.fillState = FILL_SWIRL;
						}
						else{
							fb->ShUserData.Wells[fb->ShUserData.Recipe.SampleWellCount].Present = TRUE;
							fb->ShUserData.Wells[fb->ShUserData.Recipe.SampleWellCount].Color = fb->ShUserData.Recipe.Samples[fb->ShUserData.Recipe.CurrentSample].Sample;
							fb->ShUserData.Recipe.SampleWellCount++;
							fb->ShUserData.Recipe.Samples[fb->ShUserData.Recipe.CurrentSample].CurrentCount++;
							fb->internal.fillState = FILL_CHECK_RECIPE;
						}
					}
					break;
				case FILL_SWIRL:
					if(fb->internal.fbs.moveArcFb.Done){
						fb->internal.fbs.moveArcFb.Execute = FALSE;
						fb->ShUserData.Wells[fb->ShUserData.Recipe.DyeWellCount].Color += 1;
						fb->ShUserData.Recipe.DyeWellCount++;
						fb->ShUserData.Recipe.Samples[fb->ShUserData.Recipe.CurrentSample].CurrentCount++;
						fb->internal.fillState = FILL_CHECK_RECIPE;
					}
					break;
				case FILL_CHECK_RECIPE:
					if(fb->ShUserData.Recipe.Samples[fb->ShUserData.Recipe.CurrentSample].CurrentCount == fb->ShUserData.Recipe.Samples[fb->ShUserData.Recipe.CurrentSample].SampleCount){
						//Finished filling this sample if the dye has present only (we apply the sample then the dye)
						if(fb->DyePresent){
							fb->ShUserData.Recipe.CurrentSample++;
						}
						fb->OperateDone = TRUE;
						fb->internal.state = STN_PIPETTE_WAIT_FOR_CMD;
					}
					else{
						fb->internal.fillPos.X++;
						if(fb->internal.fillPos.X == fb->WellPlateInfo.NumColumns){
							fb->internal.fbs.moveInPlaneFb.Parameters.Position.X = (fb->WellPlateInfo.NumColumns - 1)* fb->WellPlateInfo.ColumnGap;
							fb->internal.fbs.moveInPlaneFb.Parameters.Position.Y = -fb->WellPlateInfo.RowGap;
							fb->internal.fillPos.Y++;
							fb->internal.fillPos.X = 0;
						}
						else{
							fb->internal.fbs.moveInPlaneFb.Parameters.Position.X = -fb->WellPlateInfo.ColumnGap;
							fb->internal.fbs.moveInPlaneFb.Parameters.Position.Y = 0;
						}
						fb->internal.fbs.moveInPlaneFb.Execute = TRUE;
						fb->internal.fillState = FILL_MOVE;
					}
					break;
			}
			rl6dShCopyUserDataSync(&fb->internal.fbs.destMonFb.RouterShuttle,rl6dSH_COPY_USER_DATA_WRITE,&fb->ShUserData,sizeof(fb->ShUserData));
			break;
		//******************** Waiting for the send command State
		case STN_PIPETTE_WAIT_FOR_CMD:
			rl6dShCopyUserDataSync(&fb->internal.fbs.destMonFb.RouterShuttle,rl6dSH_COPY_USER_DATA_READ,&fb->ShUserData,sizeof(fb->ShUserData));
			if(fb->Send){
				//Update the user data
				rl6dShCopyUserDataSync(&fb->internal.fbs.destMonFb.RouterShuttle,rl6dSH_COPY_USER_DATA_WRITE,&fb->ShUserData,sizeof(fb->ShUserData));

				fb->internal.fbs.moveDestFb.RouterShuttle = &fb->internal.fbs.destMonFb.RouterShuttle;
				fb->internal.fbs.moveDestFb.Destination = fb->NextDestination;
				fb->internal.fbs.moveDestFb.Waypoint = fb->Waypoint;
				fb->internal.fbs.moveDestFb.Velocity = fb->Velocity;
				fb->internal.fbs.moveDestFb.Acceleration = fb->Accel;
				fb->internal.fbs.moveDestFb.Execute = TRUE;

				fb->internal.state = STN_PIPETTE_SEND;
			}
			break;
		//******************** Send Shuttle State State
		case STN_PIPETTE_SEND:
			if(fb->internal.fbs.moveDestFb.Error){
				fb->internal.errorState = fb->internal.state;
				fb->Error = TRUE;
				fb->ErrorID = fb->internal.fbs.moveDestFb.ErrorID;
				fb->internal.state = STN_PIPETTE_ERROR;
			}
			else if(fb->internal.fbs.moveDestFb.Active){
				fb->internal.fbs.destMonFb.AcknowledgeShuttle = TRUE;
				if(!fb->internal.fbs.destMonFb.ShuttlePresent){
					fb->internal.fbs.destMonFb.AcknowledgeShuttle = FALSE;
					fb->internal.fbs.moveDestFb.Execute = FALSE;
					fb->ShuttlePresent = FALSE;
					fb->WaitComplete = FALSE;
					fb->OperateDone = FALSE;
					brsmemset(&fb->ShUserData,0,sizeof(fb->ShUserData));
					brsmemset(&fb->Shuttle,0,sizeof(fb->Shuttle));
					fb->internal.state = STN_PIPETTE_DONE;
				}
			}
			break;
		//******************** Waiting for the Send Cmd To Drop State
		case STN_PIPETTE_DONE:
			if(!fb->Send){
				fb->internal.state = STN_PIPETTE_READY;
			}
			break;
		//******************** Error State
		case STN_PIPETTE_ERROR:
			if(!fb->Enable){

			}
			break;
		//******************** Reset State
		case STN_PIPETTE_RESET:

			break;
	}

	TON(&fb->internal.fbs.waitFb);
	MC_BR_MoveInPlane_Acp6D(&fb->internal.fbs.moveInPlaneFb);
	MC_BR_MoveArc_Acp6D(&fb->internal.fbs.moveArcFb);
	rl6dDestinationMonitor(&fb->internal.fbs.destMonFb);
	rl6dShuttleMoveDestination(&fb->internal.fbs.moveDestFb);
}
```

#### tipReplaceFb.c - not listed in the package file held
```c
#include <bur/plctypes.h>
#ifdef __cplusplus
	extern "C"
	{
#endif
#include "StnLogic.h"
#ifdef __cplusplus
	};
#endif

#define TRUE 1
#define FALSE 0

/* TODO: Add your comment here */
void tipReplace(struct tipReplace* fb){
	//If Tip needs replace, move to old tip
	//Move Tip Down
	//Wait
	//Move Tip up
	//Move to new tip
	//Move tip Down
	//Move Tip Up
	switch (fb->internal.state)
	{
		case TIP_IDLE:
			if(fb->Execute){
				fb->TipZPosition = fb->TipHomeZPosition;
				fb->Active = TRUE;
				fb->internal.fbs.movePlaneFb.Shuttle = fb->Shuttle;
				fb->internal.fbs.movePlaneFb.Parameters.Velocity = fb->ShuttleVel;
				fb->internal.fbs.movePlaneFb.Parameters.Acceleration = fb->ShuttleAccel;
				fb->internal.fbs.movePlaneFb.Parameters.Mode = mcACP6D_MOVE_RELATIVE;
				fb->internal.fbs.movePlaneFb.Parameters.Path = mcACP6D_PATH_DIRECT;
				fb->internal.fbs.movePlaneFb.Execute = TRUE;
				if(fb->TipNeedsReplaced){
					//Move to old tip
					fb->internal.fbs.movePlaneFb.Parameters.Position.X = fb->OldTipPosition.X;
					fb->internal.fbs.movePlaneFb.Parameters.Position.Y = fb->OldTipPosition.Y;
					fb->internal.state = TIP_MOVE_OLD;
				}
				else{
					fb->NoTip = TRUE;
					fb->internal.fbs.movePlaneFb.Parameters.Position.X = fb->NewTipPosition.X;
					fb->internal.fbs.movePlaneFb.Parameters.Position.Y = fb->NewTipPosition.Y;
					fb->internal.state = TIP_MOVE_NEW;
				}
			}
			break;
		case TIP_MOVE_OLD:
			if(fb->internal.fbs.movePlaneFb.Done){
				fb->internal.fbs.movePlaneFb.Execute = FALSE;
				fb->internal.state = TIP_LOWER_TIP;
			}
			break;
		case TIP_MOVE_NEW:
			if(fb->internal.fbs.movePlaneFb.Done){
				fb->internal.fbs.movePlaneFb.Execute = FALSE;
				fb->internal.state = TIP_LOWER_TIP;
			}
			break;
		case TIP_LOWER_TIP:
			fb->TipZPosition -= fb->TipZVelocity;
			if(fb->TipZPosition <= fb->TipZSwapHeight){
				fb->internal.fbs.waitTon.PT = fb->TipSwapTime;
				fb->internal.fbs.waitTon.IN = TRUE;

				if(fb->TipNeedsReplaced)
					fb->NoTip = !fb->NoTip;
				else
					fb->NoTip = FALSE;
				fb->internal.state = TIP_WAIT;
			}
			break;
		case TIP_RAISE_TIP:
			fb->TipZPosition += fb->TipZVelocity;

			if(fb->TipZPosition >= fb->TipHomeZPosition){
				if(!fb->internal.tipReplaced && fb->TipNeedsReplaced){
					fb->internal.tipReplaced = TRUE;
					fb->internal.fbs.movePlaneFb.Parameters.Position.X = fb->NewTipPosition.X - fb->OldTipPosition.X;
					fb->internal.fbs.movePlaneFb.Parameters.Position.Y = fb->NewTipPosition.Y;
					fb->internal.fbs.movePlaneFb.Execute = TRUE;
					fb->internal.state = TIP_MOVE_NEW;
				}
				else{
					fb->NoTip = FALSE;
					fb->Done = TRUE;
					fb->internal.state = TIP_DONE;
				}
			}
			break;
		case TIP_WAIT:
			if(fb->internal.fbs.waitTon.Q){
				fb->internal.fbs.waitTon.IN = FALSE;
				fb->internal.state = TIP_RAISE_TIP;
			}
			break;
		case TIP_DONE:
			if(!fb->Execute){
				fb->Active = FALSE;
				fb->Done = FALSE;
				fb->internal.tipReplaced = FALSE;
				fb->internal.state = TIP_IDLE;
			}
			break;
	}
	MC_BR_MoveInPlane_Acp6D(&fb->internal.fbs.movePlaneFb);
	TON(&fb->internal.fbs.waitTon);
}
```


### Program Logical/Source/ScnViewer/Vis (IEC)

#### Types.typ
```iecst
TYPE
	VisTyp : 	STRUCT
		Shuttles : ARRAY[0..MAX_SH_IDX]OF ShuttleVisTyp;
	END_STRUCT;
	ShuttleVisTyp : 	STRUCT
		Visible : BOOL;
		Position : VisPositionTyp;
		ShuttleColor : ColorEnum;
		Wells : ARRAY[0..17]OF WellTyp;
		ToolVisible : BOOL;
	END_STRUCT;
	VisPositionTyp : 	STRUCT
		X : REAL;
		Y : REAL;
		Z : REAL;
	END_STRUCT;
END_TYPE
```

#### Variables.var
```iecst
VAR
	userData : UserDataType;
	i : USINT;
	Vis : VisTyp;
	shInfoFB : ARRAY[0..MAX_SH_IDX] OF MC_BR_ShReadInfo_Acp6D;
END_VAR
```

#### Cyclic.st
```iecst
PROGRAM _CYCLIC
	FOR i := 0 TO MAX_SH_IDX DO
		IF gShIfs[i].Cfg.Shuttle.controlif <> 0 THEN
			Vis.Shuttles[i].Visible := TRUE;
			shInfoFB[i].Enable := TRUE;
			shInfoFB[i].Shuttle := ADR(gShIfs[i].Cfg.Shuttle);

			shInfoFB[i]();
			Vis.Shuttles[i].Position.X := shInfoFB[i].ShuttleInfo.Position.X * 1000;
			Vis.Shuttles[i].Position.Y := shInfoFB[i].ShuttleInfo.Position.Y * 1000;
			Vis.Shuttles[i].Position.Z := shInfoFB[i].ShuttleInfo.Position.Z * 1000;

			IF gShIfs[i].Cfg.RouterShuttle.Ident <> 0 AND i < 3 THEN
				rl6dShCopyUserDataSync(gShIfs[i].Cfg.RouterShuttle,rl6dSH_COPY_USER_DATA_READ,ADR(userData),SIZEOF(userData));
				Vis.Shuttles[i].Wells := userData.Wells;
				Vis.Shuttles[i].ShuttleColor := userData.CurrentColor;
				IF Vis.Shuttles[i].ShuttleColor = COLOR_UNDEF THEN
					Vis.Shuttles[i].ToolVisible := FALSE;
				ELSE
					Vis.Shuttles[i].ToolVisible := TRUE;
				END_IF
			END_IF
		ELSE
			Vis.Shuttles[i].Visible := FALSE;
			shInfoFB[i].Enable := FALSE;
			shInfoFB[i]();
		END_IF
	END_FOR;

END_PROGRAM
```

#### Init.st
```iecst
PROGRAM _INIT

END_PROGRAM
```

- BuildVersion.ps1 (not shown)

- Visualisation Logical/mappView (not shown)

Listed in the project but not available here: Logical/Source/Core/StnLogic/Constants.var
